	IF(inResult.Result<>eOverallResult.Failed ) THEN
		THIS^.StationBase.RecurringFails.AnyRecurringFails.Counter:=0;
		THIS^.StationBase.RecurringFails.AnyRecurringFails.Reached :=FALSE;
		This^.CompleteStep();
	ELSE
		//collect any recurring fails
		IF NOT THIS^.StationBase.RecurringFails.AnyRecurringFails.Reached THEN 
			THIS^.StationBase.RecurringFails.AnyRecurringFails.Counter := THIS^.StationBase.RecurringFails.AnyRecurringFails.Counter +1;
		END_IF
		THIS^.StationBase.RecurringFails.AnyRecurringFails.Reached:=THIS^.StationBase.RecurringFails.AnyRecurringFails.Counter>=THIS^.StationBase._settings.AnyRecurringFailure;
		

		
	

		
		THIS^.Messenger.OnCondition(THIS^.StationBase.RecurringFails.AnyRecurringFails.Reached)
									   .Build()
									   .Append('(Consecutive failure) The number of any recurring failure count has been reached!')
									   .Append(' Failure code: ')
									   .Append(inResult.ErrorCodes)
  									   .Append(' ')
									   .Append(inResult.Failures)						
									   .As()				   
									   .AsError();
									   
		THIS^.StepCompleteWhen(NOT THIS^.StationBase.RecurringFails.AnyRecurringFails.Reached);			
						   
									   
		IF THIS^.StationBase.RecurringFails.AnyRecurringFails.Reached THEN
			
				
			IF(_dialog.Show()
			   .WithCaption('<#(Consecutive failure) The number of any recurring failure count has been reached!#>')
			   .WithText('<#Please acknowledge recurring failure!#>')
			   .WithOk().Answer = TcoCore.eDialogAnswer.OK) THEN
			   
					THIS^.StationBase.RecurringFails.AnyRecurringFails.Counter:=0;
					THIS^.StationBase.RecurringFails.AnyRecurringFails.Reached :=FALSE;
					THIS^.CompleteStep();
			END_IF; 
		END_IF;
	END_IF;
	

	
	
	
 		    				
    //-------------------------------------
END_IF
END_METHOD

METHOD MonitorSameRecurringFailure
VAR_INPUT
	(*~
	<docu>
		<summary>
			The unique step id definition.
		</summary>			
	</docu>	
	~*)
	inStepID : INT;
		(*~
	<docu>
		<summary>
			The step enable condition.
		</summary>			
	</docu>	
	~*)
	inEnableStep :BOOL;
	inResult : TcoComprehensiveResult;
END_VAR
IF (Step(inStepID,inEnableStep, 'MONITOR SAME RECURRING FAILURE IN SEQUENCE')) THEN
    //-------------------------------------		
	
	IF(inResult.Result<>eOverallResult.Failed ) THEN
		THIS^.StationBase.RecurringFails.SameRecurringFails.Counter:=0;
		THIS^.StationBase.RecurringFails.SameRecurringFails.Reached :=FALSE;
		THIS^.CompleteStep();
	ELSE
	
		//collect same recurring
		IF NOT THIS^.StationBase.RecurringFails.SameRecurringFails.Reached THEN 
			IF THIS^.StationBase.RecurringFails.SameRecurringFails.Result.ErrorCodes = inResult.ErrorCodes AND inResult.ErrorCodes <>';' THEN //if error code not defined ignore
				THIS^.StationBase.RecurringFails.SameRecurringFails.Counter := THIS^.StationBase.RecurringFails.SameRecurringFails.Counter +1;
			END_IF;
			THIS^.StationBase.RecurringFails.SameRecurringFails.Result.ErrorCodes := inResult.ErrorCodes ;
		END_IF;
		
		THIS^.StationBase.RecurringFails.SameRecurringFails.Reached:=THIS^.StationBase.RecurringFails.SameRecurringFails.Counter>=THIS^.StationBase._settings.SameRecurringFailure;

			
		THIS^.Messenger.OnCondition(THIS^.StationBase.RecurringFails.SameRecurringFails.Reached)
									   .Build()
									   .Append('(Consecutive failure) The number of same recurring failure count has been reached!')
									   .Append(' Failure code: ')
									   .Append(inResult.ErrorCodes)
  									   .Append(' ')
									   .Append(inResult.Failures)									   									   
									   .As()				   
									   .AsError();
		
		THIS^.StepCompleteWhen(NOT THIS^.StationBase.RecurringFails.SameRecurringFails.Reached);
	

									   
		IF THIS^.StationBase.RecurringFails.SameRecurringFails.Reached THEN
			IF(_dialog.Show()
			   .WithCaption('<#(Consecutive failure) The number of same recurring failure count has been reached!#>')
			   .WithText('<#Please acknowledge recurring failure!#>')
			   .WithOk().Answer = TcoCore.eDialogAnswer.Ok) THEN
			   
					THIS^.StationBase.RecurringFails.SameRecurringFails.Counter:=0;
					THIS^.StationBase.RecurringFails.SameRecurringFails.Reached :=FALSE;
					THIS^.CompleteStep();
			END_IF; 
		END_IF
	END_IF;
	

	
	
	
 		    				
    //-------------------------------------
END_IF
END_METHOD

PROPERTY StationBase : REFERENCE TO CuBase
GET
VAR
    _station : POINTER TO CUBase;
END_VAR
IF __QUERYPOINTER(Parent, _station) THEN // Check if _Parent is Station001
    StationBase REF= _station^;              // If the check is successful dereference a pointer. simlar to THIS^ or SUPER^
END_IF
END_GET
END_PROPERTY

END_FUNCTION_BLOCK

// ---- Abstractions/TcoCore/TcoTaskedSequencer.TcPOU
FUNCTION_BLOCK PUBLIC ABSTRACT TcoTaskedSequencer EXTENDS TcoCore.TcoSequencerBase
VAR
	{attribute addProperty Name "|[[1]AttributeName]|"}
	{attribute addProperty ToolTip "|[[1]AttributeToolTip]|"}
    _task : TcoInnerTask(THIS^);
    _o    : TcoCore.TcoSequencerObserver(THIS^);	
	{attribute addProperty Name "|[[1]Cycle Time Analitics]|"} 
	_cycleTimeAnalitics:CycleTimeAnalitics;	
	_startCleanCycleTime: TIME;
	_stopCleanCycleTime: TIME;
	_timer_1: TON;
	_timer_2: TON;
END_VAR

Run();

PROPERTY PUBLIC AverageCleanCycleTime : TIME
GET
AverageCleanCycleTime:=_cycleTimeAnalitics.AverageCleanCycle;
END_GET
END_PROPERTY

PROPERTY PUBLIC AverageCycleTime : TIME
GET
AverageCycleTime:=_cycleTimeAnalitics.Average;
END_GET
END_PROPERTY

(*~
	<docu>
		<summary>
			Completes the actually running step, when the `inCondition` parameter is `TRUE`.
			Method is typically called inside a step as the transition method.
		</summary>			
	</docu>	
~*)
METHOD PROTECTED FINAL Await
VAR_INPUT
    (*~
	<docu>
		<summary>
			The condition under which the step is completed.
		</summary>			
	</docu>	
~*)
    inCondition : BOOL;
END_VAR
i_StepCompleteWhen(inCondition := inCondition);
END_METHOD

(*~
	<docu>
		<summary>
			<para>
				Completes the sequencer, and return the sequencer pointer to the first step in the seuqence.
				Method is typically called inside the last step of the sequence.
			</para>
		</summary>			
	</docu>	
~*)
METHOD PROTECTED FINAL CompleteSequence
i_CompleteSequence();

IF _cycleTimeAnalitics.FilterConstant = 0 THEN;
	_cycleTimeAnalitics.FilterConstant:=10;
END_IF;


IF _cycleTimeAnalitics.Average = T#0S THEN
	_cycleTimeAnalitics.Average:=_SequenceElapsedTime;
END_IF
_cycleTimeAnalitics.Average:= (((_cycleTimeAnalitics.FilterConstant-1)*_cycleTimeAnalitics.Average)+_LastCycleTime)/_cycleTimeAnalitics.FilterConstant;

_startCleanCycleTime:=T#0S;
_stopCleanCycleTime:=T#0S;
END_METHOD

(*~
	<docu>
		<summary>
			Completes the execution of the current step and moves the sequencer pointer to the next step in order of execution.
			The call returns `ITcoObjectRestorer` that allows to restore object upon step completition.
		</summary>		
		<returns></returns>	
	</docu>	
~*)
METHOD PROTECTED FINAL CompleteStep : ITcoObjectRestorer
CompleteStep := i_CompleteStep();
END_METHOD

PROPERTY PUBLIC CycleTimeFilterConstant : UINT
GET
CycleTimeFilterConstant:=_cycleTimeAnalitics.FilterConstant;
END_GET
SET // PUBLIC
_cycleTimeAnalitics.FilterConstant:=CycleTimeFilterConstant;
END_SET
END_PROPERTY

(*~
	<docu>
		<summary>
			Main method of the sequener. Custom code needs to be placed here. The sequencer is executed by call of **Instance.Run()** method.
			This method is abstract, and it must be overridden in derived block.
		</summary>
	</docu>
~*)
METHOD PROTECTED  Main : BOOL
END_METHOD

METHOD PUBLIC OnAbort : BOOL
SUPER^.Restore();
END_METHOD

METHOD PUBLIC OnDone : BOOL
END_METHOD

METHOD PUBLIC OnError : BOOL
END_METHOD

METHOD PUBLIC OnStart
_startCleanCycleTime:=T#0S;
_stopCleanCycleTime:=T#0S;
END_METHOD

METHOD pr_Close
VAR_INPUT
END_VAR
_lastClosingCycle := Context.StartCycleCount;

IF _sequencerHasError THEN
    OnSequencerError(_sequencerErrorId);
END_IF

_previousNumberOfStepsInSequence := _numberOfStepsInSequence;
Context.Environment.Messaging.Suspend();

IF _modeController._stepIn.Done THEN
    _modeController._stepIn.Restore();
END_IF

Context.Environment.Messaging.Resume();

_restoringSequence := FALSE;
END_METHOD

METHOD pr_Open
VAR
    _message : STRING(255);
END_VAR
_theOrderOfTheCurrentlyEvaluatedStep := 0;

IF _requestStepActive AND
    _requestedStepId <> (MinStepID - 1) AND
    (_modeController.Mode <> eSequencerMode.StepMode OR _modeController._stepIn.Busy OR _checkStepIdRequestedInStepMode) THEN
    _requestStepCycle := _requestStepCycle + 1;
ELSE
    _requestStepCycle := 0;
END_IF

IF _requestStepCycle > 1 AND NOT _sequencerHasError THEN
    _sequencerErrorId        := eSequencerError.StepWithRequestedIdDoesNotExists;
    _message                 := CONCAT('REQUESTED STEP_ID: ', INT_TO_STRING(_requestedStepId));
    _message                 := CONCAT(_message, ' DOES NOT EXIST');
    _currentStep.Description := _message;
    _currentStep.Status      := eStepStatus.Error;
    THIS^.Messenger.Post(_message, eMessageCategory.ProgrammingError);
    _sequencerHasError := TRUE;
END_IF

IF _StepIdUniquenessControlState = eStepIdUniquenessControlState.NotYetStarted OR
    _StepIdUniquenessControlState = eStepIdUniquenessControlState.Requested THEN
    _StepIdUniquenessControlState := eStepIdUniquenessControlState.Started;
END_IF;

_restoringSequence := FALSE;

_lastOpeningCycle := Context.StartCycleCount;
;
END_METHOD

(*~
	<docu>
		<summary>
			Terminates the currently executed step and set the sequencer's pointer to the step with Id that corresponds to ```inRequestedStepID``` parameter.
			When the order of the requested step is higher than the order of the currently finished step (the requested step is "after" the current one)
			the requested step is started in the same context cycle.
			When the order of the requested step is lower than the order of the currently finished step (the requested step is "before" the current one)
			the requested step is started in the next context cycle.
			If the requested step is not found even in the next context cycle, the sequencer enters error state ```StepWithRequestedIdDoesNotExists```.
			<para>
				See <see cref="TcoCore.eSequencerError"/> for detailed description.
			</para>
		</summary>
	</docu>
~*)
METHOD PROTECTED FINAL RequestStep : ITcoSequencer
VAR_INPUT
    (*~
		<docu>
			<summary>
				StepId of the step to be executed.
			</summary>
		</docu>
	~*)
    inRequestedStepID : INT := MinStepID - 1;
END_VAR
VAR
    _message : STRING(254);
END_VAR
RequestStep := i_RequestStep(inRequestedStepID := inRequestedStepID);
END_METHOD

(*~
	<docu>
		<summary>
			This method resets the sequencer cycle time . 
				Method is typically called before starting the sequence(e.g.in ground position task) .
		</summary>		
		<returns></returns>	
	</docu>	
~*)
METHOD PUBLIC ResetCycleTime
VAR_INPUT
END_VAR

_cycleTimeAnalitics.Average:=T#0S;
_cycleTimeAnalitics.AverageCleanCycle:=T#0S;
END_METHOD

METHOD PRIVATE ResetTimers
VAR_INPUT
END_VAR
_timer_1.IN:=FALSE;
_timer_2.IN:=FALSE;
END_METHOD

(*~
	<docu>
		<summary>
			<para>
				This method resets the sequencer. 
				Method is typically called before starting the sequence or after error has occured in the sequence.
			</para>
		</summary>			
	</docu>	
~*)
METHOD PUBLIC Restore : ITcoRestorable
SUPER^.Restore();
Task.Restore();
END_METHOD

(*~
	<docu>
		<summary>
			<para>
				Ensures calling the Open(), Main() and Close() methods in the desired order.
				This method is final, so it cannot be overloaded. The **Instance.Run()** needs to be called cyclically inside the appropriate context.
			</para>
		</summary>			
	</docu>	
~*)
METHOD PUBLIC FINAL Run
VAR
    _message : STRING;
END_VAR
IF (_task.Execute()) THEN
    THIS^.pr_Open();
    THIS^.Observer := _o;
    THIS^.Main();
    THIS^.pr_Close();
END_IF;
END_METHOD

(*~
	<docu>
		<summary>
			This method s used to start the clean cycle time measurement . 
				Method is typically called at the beggining of the sequence(e.g.in automat sequence) .
		</summary>		
		<returns></returns>	
	</docu>	
~*)

METHOD PUBLIC StartCleanCycleTime
VAR_INPUT
END_VAR
_stopCleanCycleTime:=t#0s;
_startCleanCycleTime:=_SequenceElapsedTime;
END_METHOD

METHOD PROTECTED Step : BOOL
VAR_INPUT
    (*~
	<docu>
		<summary>
			StepId of the current step.
			<remarks>			
				<note type="important">
					This number must be unique throughout the complete sequence.
					It must be a constant or numerical literal and it must not change during the life-time of the sequencer. 
				</note>
			</remarks>
		</summary>		
	</docu>	
~*)
    inStepID : INT;
    (*~
	<docu>
		<summary>
			If this value is false, step body is not executed and execution is moved to the next enabled step.
		</summary>				
	</docu>	
~*)
    inEnabled : BOOL;
    (*~
	<docu>
		<summary>
			Step description text.
		</summary>				
	</docu>	
~*)
    inStepDescription : STRING(254);
END_VAR
Step := i_Step(inStepID := inStepID, inEnabled := inEnabled, inStepDescription := inStepDescription);
END_METHOD

(*~
	<docu>
		<summary>
			Completes the actually running step, when the `inCondition` parameter is `TRUE`.
			Method is typically called inside a step as the transition method.
		</summary>			
	</docu>	
~*)
METHOD PROTECTED FINAL StepCompleteWhen
VAR_INPUT
    (*~
	<docu>
		<summary>
			The condition under which the step is completed.
		</summary>			
	</docu>	
~*)
    inCondition : BOOL;
END_VAR
i_StepCompleteWhen(inCondition := inCondition);
END_METHOD

(*~
	<docu>
		<summary>
			This method s used to stop the clean cycle time measurement . 
				Method is typically called at the end of the sequence(e.g.in automat sequence )  .
		</summary>		
		<returns></returns>	
	</docu>	
~*)

METHOD PUBLIC StopCleanCycleTime
VAR_INPUT
END_VAR

VAR
	cleanCycleTime: TIME;
END_VAR
_stopCleanCycleTime:=_SequenceElapsedTime;

cleanCycleTime:=T#0S;
IF _stopCleanCycleTime>_startCleanCycleTime THEN
	cleanCycleTime:=_stopCleanCycleTime-_startCleanCycleTime;
 END_IF;

IF _cycleTimeAnalitics.FilterConstant = 0 THEN;
	_cycleTimeAnalitics.FilterConstant:=10;
END_IF;


IF _cycleTimeAnalitics.AverageCleanCycle = T#0S THEN
	_cycleTimeAnalitics.AverageCleanCycle:=_stopCleanCycleTime;
END_IF
_cycleTimeAnalitics.AverageCleanCycle:= (((_cycleTimeAnalitics.FilterConstant-1)*_cycleTimeAnalitics.AverageCleanCycle)+cleanCycleTime)/_cycleTimeAnalitics.FilterConstant;
END_METHOD

PROPERTY Task : REFERENCE TO TcoTask
GET
Task REF= _task;
END_GET
END_PROPERTY

METHOD PUBLIC FINAL Timer_1 : BOOL
VAR_INPUT
	Condition : BOOL;
	PT : TIME;
END_VAR
_timer_1(IN:= Condition  and  not IsFreshState, PT:=PT);
Timer_1 := _timer_1.Q;
END_METHOD

METHOD PUBLIC FINAL Timer_2 : BOOL
VAR_INPUT
	Condition : BOOL;
	PT : TIME;
END_VAR
_timer_2(IN:= Condition and not IsFreshState, PT:=PT);
Timer_2 := _timer_2.Q;
END_METHOD

END_FUNCTION_BLOCK

// ---- Abstractions/TcoCore/TcoInnerTask.TcPOU
FUNCTION_BLOCK TcoInnerTask EXTENDS TcoCore.TcoTask

(*~
	<docu>
		<summary>
			Executes when task is aborted.
		</summary>			
	</docu>	
~*)
METHOD PROTECTED OnAbort
ParentSequencer.OnAbort();
END_METHOD

(*~
	<docu>
		<summary>
			Executes when task reaches the ```Done``` state .
		</summary>			
	</docu>	
~*)
METHOD PROTECTED OnDone
ParentSequencer.OnDone();
END_METHOD

(*~
	<docu>
		<summary>
			Executes when task reaches the ```Error``` state.
			<para>
				Do not confuse with <see cref="PlcDocu.TcoCore.TcoTask.WhileError()"/>, that is called cyclically until '''Error''' state is left.
			</para>
		</summary>			
	</docu>	
~*)
METHOD PROTECTED OnError
ParentSequencer.OnError();
END_METHOD

METHOD PROTECTED OnStart
ParentSequencer.OnStart();
END_METHOD

PROPERTY PRIVATE ParentSequencer : REFERENCE TO TcoTaskedSequencer
GET
VAR
	_sequencer : POINTER TO TcoTaskedSequencer;
END_VAR
IF __QUERYPOINTER(Parent, _sequencer) THEN // Check if _Parent is Station001
    ParentSequencer REF= _sequencer^;              // If the check is successful dereference a pointer. simlar to THIS^ or SUPER^
END_IF
END_GET
END_PROPERTY

END_FUNCTION_BLOCK

// ---- Abstractions/CUBase/Tasks/CUBaseGround.TcPOU
FUNCTION_BLOCK ABSTRACT CUBaseGround EXTENDS TcoTaskedSequencer
VAR
	_groundDone : BOOL;
END_VAR

METHOD INTERNAL CancelGround
_groundDone := FALSE;
END_METHOD

PROPERTY GroundDone : BOOL
GET
GroundDone := _groundDone;
END_GET
END_PROPERTY

END_FUNCTION_BLOCK

// ---- Abstractions/TcoCore/TcoTaskedService.TcPOU
FUNCTION_BLOCK PUBLIC ABSTRACT TcoTaskedService EXTENDS TcoCore.TcoTask
VAR
	
END_VAR

(*~
	<docu>
		<summary>
			Main method of the sequener. Custom code needs to be placed here. The sequencer is executed by call of **Instance.Run()** method.
			This method is abstract, and it must be overridden in derived block.
		</summary>
	</docu>
~*)
METHOD PROTECTED ABSTRACT Main : BOOL
END_METHOD

(*~
	<docu>
		<summary>
			<para>
				Ensures calling the Open(), Main() and Close() methods in the desired order.
				This method is final, so it cannot be overloaded. The **Instance.Run()** needs to be called cyclically inside the appropriate context.
			</para>
		</summary>			
	</docu>	
~*)
METHOD PUBLIC FINAL Run
VAR
    _message : STRING;
END_VAR
IF (THIS^.Execute()) THEN
    THIS^.Main();    
END_IF;
END_METHOD

PROPERTY Task : REFERENCE TO TcoTask
GET
Task REF= THIS^;
END_GET
END_PROPERTY

END_FUNCTION_BLOCK

// ---- Abstractions/CUBase/Tasks/CUBaseRecover.TcPOU
FUNCTION_BLOCK ABSTRACT CUBaseRecover EXTENDS TcoTaskedSequencer
VAR
	_done:BOOL;

END_VAR

PROPERTY Done : bool
GET
Done := _done;
END_GET
END_PROPERTY

METHOD PUBLIC OnStart
_done:=FALSE;
END_METHOD

PROPERTY StationBase : REFERENCE TO CuBase
GET
VAR
    _station : POINTER TO CuBase;
END_VAR
IF __QUERYPOINTER(Parent, _station) THEN // Check if _Parent is Station001
    StationBase REF= _station^;              // If the check is successful dereference a pointer. simlar to THIS^ or SUPER^
END_IF
END_GET
END_PROPERTY

END_FUNCTION_BLOCK

// ---- Abstractions/CUBase/Tasks/CUBaseSuspend.TcPOU
FUNCTION_BLOCK ABSTRACT CUBaseSuspend EXTENDS TcoTaskedSequencer
VAR
	_done:BOOL;

END_VAR

PROPERTY Done : bool
GET
Done := _done;
END_GET
END_PROPERTY

METHOD PUBLIC OnStart
_done:=FALSE;
END_METHOD

PROPERTY StationBase : REFERENCE TO CuBase
GET
VAR
    _station : POINTER TO CuBase;
END_VAR
IF __QUERYPOINTER(Parent, _station) THEN // Check if _Parent is Station001
    StationBase REF= _station^;              // If the check is successful dereference a pointer. simlar to THIS^ or SUPER^
END_IF
END_GET
END_PROPERTY

END_FUNCTION_BLOCK

// ---- Technology/CU00x/Manual/CU00xManualTask.TcPOU
FUNCTION_BLOCK CU00xManualTask EXTENDS TcoTaskedService IMPLEMENTS ICUTask
VAR
END_VAR

Run();

(*~
	<docu>
		<summary>
			Main method of the sequener. Custom code needs to be placed here. The sequencer is executed by call of **Instance.Run()** method.
			This method is abstract, and it must be overridden in derived block.
		</summary>
	</docu>
~*)
METHOD PROTECTED Main : BOOL
Messenger.Notify('Running manual mode');
// Station.Components.OUT1.Service();
// Station.Components.OUT2.Service();
// Station.Components.OUT3.Service();
END_METHOD

METHOD PROTECTED OnStart
Station.AutomatTask.Restore();
Station.GroundTask.Restore();
Station.GroundTask.CancelGround();
END_METHOD

PROPERTY Station : REFERENCE TO CU00x
GET
VAR
    _station : POINTER TO CU00x;
END_VAR
IF __QUERYPOINTER(Parent, _station) THEN // Check if _Parent is Station001
    Station REF= _station^;              // If the check is successful dereference a pointer. simlar to THIS^ or SUPER^
END_IF
END_GET
END_PROPERTY

END_FUNCTION_BLOCK

// ---- Technology/CU00x/Ground/CU00xGroundTask.TcPOU
FUNCTION_BLOCK CU00xGroundTask EXTENDS CUBaseGround IMPLEMENTS ICUTask

Run();

METHOD DataEntityDiscard
VAR_INPUT	
	inStepID : INT;
	EntityId : STRING(255);
END_VAR
IF (Step(inStepID, TRUE, 'DISCARD ENTITY')) THEN	
    //-------------------------------------		
	IF(Station.ProcessDataManager.Exists(EntityId).Done) THEN
		IF(Station.ProcessDataManager._idExistsTask.Exists) THEN
			StepCompleteWhen(THIS^.Station.EntityFlowDiscard(EntityId, Station.ProcessDataManager.Data.CU00x.Header).Done);
		ELSE
			CompleteStep();
		END_IF
	END_IF;					   		    				
    //-------------------------------------
END_IF
END_METHOD

(*~
	<docu>
		<summary>
			Main method of the sequener. Custom code needs to be placed here. The sequencer is executed by call of **Instance.Run()** method.
			This method is abstract, and it must be overridden in derived block.
		</summary>
	</docu>
~*)
METHOD PROTECTED Main : BOOL
IF (Step(100, TRUE, 'STOPPING OTHER MODES')) THEN
	Station.AutomatTask.ResetCycleTime();//here we can reset averages values of CT
	Station.AutomatTask.Restore();
	Station.ManualTask.Restore();
	Station.ProcessDataManager.Restore();
	Station.AutomatTask.HideAllDialogs();
	Station.GroupInspection.Restore();// hide all dialogs 
    StepCompleteWhen(TRUE);
END_IF

IF (Step(200, TRUE, 'STOPPING OTHER MODES')) THEN	
//	---------------------------------------------------
	
	Station.AutomatTask.ResetCycleTime();
	Station.ProductionPlanerTask.Restore();
	
	Messenger.Info('INFO MESSAGE');
	
    StepCompleteWhen(THIS^._currentStep.Duration > T#500MS);
//	---------------------------------------------------
END_IF

DataEntityDiscard(5000, THIS^.Station.ProcessDataManager.Data._EntityId);

IF (Step(10000, TRUE, 'LAST STEP')) THEN	
	//---------------------------------------------------
	_groundDone := TRUE;
	THIS^._task.DoneWhen(_groundDone);
	//---------------------------------------------------
END_IF
END_METHOD

METHOD PUBLIC OnStart
SUPER^.OnStart();
Station.AutomatTask.Restore();
Station.ManualTask.Restore();
Station.GroundTask.CancelGround();
END_METHOD

PROPERTY Station : REFERENCE TO CU00x
GET
VAR
    _station : POINTER TO CU00x;
END_VAR
IF __QUERYPOINTER(Parent, _station) THEN // Check if _Parent is Station001
    Station REF= _station^;              // If the check is successful dereference a pointer. simlar to THIS^ or SUPER^
END_IF
END_GET
END_PROPERTY

END_FUNCTION_BLOCK

// ---- Technology/CU00x/Automat/CU00xAutomatTask.TcPOU
FUNCTION_BLOCK CU00xAutomatTask EXTENDS CUBaseAutomat IMPLEMENTS ICUTask
VAR

    _missingProcessSettingMessage : TcoCore.TcoMessenger(THIS^);
    _paralellTask : CU00xAutomatParalell_1_Task(THIS^, TcoCore.eRestoreMode.None);

    _sb : TcoCore.StringBuilder;

    _customizedContentInput : CU00xDialogContent(THIS^);
END_VAR

VAR
    _dataLoadProcessSettings : BOOL;
    _dataLoadProcessSettingsByPlaner : BOOL;
    _dataCreateNew : BOOL;
    _dataOpen : BOOL;
    _dataClose : BOOL;
    _dataFinalize : BOOL;
    _continueRestore : BOOL;
    _loop : BOOL;
    _inspectionResult : BOOL;
    _inspectionDimensionResult : REAL;
    _reqKey : STRING;
    _reqAssignedValue : STRING;
    _inspectorSingleExamples : BOOL;
    _inspectorGroupExamples : BOOL;
	_dialogExamples : BOOL;

END_VAR

Run();

(*~
	<docu>
		<summary>
			Loads technology settings from the current technology set into this controlled unit.
			The `StationProcessDataManager.Data` is populated by data from process settings.						
		</summary>
	</docu>
~*)
METHOD DataLoadProcessSettings : BOOL
VAR_INPUT
	inStepID : INT;
END_VAR

VAR
	_ans: TcoCore.eDialogAnswer;
END_VAR
IF (Step(inStepID, _dataLoadProcessSettings, 'LOAD PROCESS SETTING')) THEN
    //-------------------------------------
	
	THIS^._missingProcessSettingMessage.OnCondition(Station.Technology.ProcessSettings.Data._EntityId = '')
									   .Build()
									   .Append('No process data. Please load setting')
									   .As()				   
									   .AsError()
									   .Pin();
					   
				   
	IF(Station.Technology.ProcessSettings.Data._EntityId <> '' (*AND NOT THIS^._missingProcessSettingMessage.Pinned*)) THEN
		IF(Station.Technology.ProcessSettings.Read(Station.Technology.ProcessSettings.Data._EntityId).Done) THEN
			Station.ProcessDataManager.Data := Station.Technology.ProcessSettings.Data;
			Station.ProcessDataManager.Data.EntityHeader.RecipeCreated := Station.Technology.ProcessSettings.Data._Created;
			Station.ProcessDataManager.Data.EntityHeader.RecipeLastModified  := Station.Technology.ProcessSettings.Data._Modified;
			Station.ProcessDataManager.Data.EntityHeader.Recipe  := Station.Technology.ProcessSettings.Data._EntityId;				
			CompleteStep();

		END_IF;	
	ELSE
		_ans:=_dialog.Show()
			.WithImage('d:\MTS\Develop\TcOpenGroup\TcOpen\assets\logo\TcOpenWide.png',400,600)	
	       .WithCaption('<#Process data not selected#>')
		   .WithText('<#Would you like to load default settings?#>')
		   .WithYesNoCancel().Answer;
		IF(_ans=TcoCore.eDialogAnswer.Cancel) THEN
			this^.Restore();
		END_IF
		IF( _ans= TcoCore.eDialogAnswer.Yes) THEN
		   
		   	Station.Technology.ProcessSettings.Data._EntityId := 'default';
		END_IF; 

			
	END_IF		    				
    //-------------------------------------
END_IF
END_METHOD

(*~
	<docu>
		<summary>
			Loads process settings from the current process set into this controlled unit.
			The `StationProcessDataManager.Data` is populated by data from process settings.						
		</summary>
	</docu>
~*)
METHOD DataLoadProcessSettingsByPlaner : BOOL
VAR_INPUT
	inStepID : INT;
END_VAR
IF (Step(inStepID, _dataLoadProcessSettingsByPlaner, 'LOAD PROCESS SETTING BY THE PRODUCTION PLANER')) THEN
    //-------------------------------------


								   
	 IF Station.ProductionPlanerTask.Invoke().Done	AND_THEN(Station.ProductionPlanerTask.RequiredProcessSettingsId <> '') THEN
		
		IF NOT Station.ProductionPlanerTask.ProductionPlanCompleted and_then (Station.Technology.ProcessSettings.Read(Station.ProductionPlanerTask.RequiredProcessSettingsId).Done)
			 THEN
			Station.ProcessDataManager.Data := Station.Technology.ProcessSettings.Data;
			Station.ProcessDataManager.Data.EntityHeader.RecipeCreated := Station.Technology.ProcessSettings.Data._Created;
			Station.ProcessDataManager.Data.EntityHeader.RecipeLastModified  := Station.Technology.ProcessSettings.Data._Modified;
			Station.ProcessDataManager.Data.EntityHeader.Recipe  := Station.Technology.ProcessSettings.Data._EntityId;				
			CompleteStep();
			Station.ProductionPlanerTask.Restore();
		END_IF;
	ELSIF  Station.ProductionPlanerTask.ProductionPlanIsEmpty THEN
		IF (_dialog.Show()
	       .WithCaption('<#Production planer#>')
		   .WithText('<#Production planer is empty!#>')
			.WithOk().Answer = TcoCore.eDialogAnswer.OK) THEN;
			;// Production plan comleted , here you can write diferent scenario ( leave it with current state , provide ground etc)	 
	
		 	//Station.GroundTask.Task.Invoke();
		   
		End_if;
	
	ELSIF  Station.ProductionPlanerTask.ProductionPlanCompleted THEN
		IF (_dialog.Show()
	       .WithCaption('<#Production planer#>')
		   .WithText('<#Production planer completed required plan!#>')
			.WithOk().Answer = TcoCore.eDialogAnswer.OK) THEN;
			;// Production plan comleted , here you can write diferent scenario ( leave it with current state , provide ground etc)	 
	
		 	//Station.GroundTask.Task.Invoke();
		   
		End_if;

			
	END_IF		    				
    //-------------------------------------
END_IF
END_METHOD

METHOD DialogExamples
VAR_INPUT
		inStepID : INT;
END_VAR
IF (Step(inStepID, TRUE, 'DIALOG EXAMPLE ')) THEN
//-------------------------------------
		_dialog.Show()
            .WithType(eDialogType.Question)
            .WithYesNo()
            .WithCaption('Hey')
            .WithText('Do we go ahead ');

        IF (_dialog.Answer = TcoCore.eDialogAnswer.Yes) THEN
            CompleteStep();
        END_IF;

        IF (_dialog.Answer = TcoCore.eDialogAnswer.No) THEN
            ;
        END_IF;

//-------------------------------------
END_IF;

IF (Step(inStepID+10, TRUE, 'DIALOG EXAMPLE WIT IMAGE')) THEN
//-------------------------------------
		_dialog.Show()
            .WithType(eDialogType.Question)
            .WithYesNo()
			.WithImage('D:\MTS\Develop\TcOpenGroup\TcOpen\assets\logo\TcOpenLogo.png',400,600)
            .WithCaption('Hey 1')
            .WithText('Do we go ahead ?');

        IF (_dialog.Answer = TcoCore.eDialogAnswer.Yes) THEN
            CompleteStep();
        END_IF;

        IF (_dialog.Answer = TcoCore.eDialogAnswer.No) THEN
            ;
        END_IF;

//-------------------------------------
END_IF;


IF (Step(inStepID+20, TRUE, 'DIALOG EXAMPLE WITH CLOSE FROM PLC')) THEN
//-------------------------------------
		_dialog.ShowWithExternalClose(inOkAnswerSignal:=FALSE , inYesAnswerSignal:= CurrentStep.Duration>T#2000MS, inNoAnswerSignal:= FALSE, inCancelAnswerSignal:= FALSE)
		    .WithType(eDialogType.Info)
            .WithYesNoCancel()
            .WithCaption('Hey')
            .WithText('Do you wana retry it? Yes answer will be set in 4 sec?');

        IF (_dialog.Answer = TcoCore.eDialogAnswer.Yes) THEN
            CompleteStep();
        END_IF;

      

//-------------------------------------
END_IF;

IF (Step(inStepID+30, TRUE, 'CUSTOMIZED DIALOG EXAMPLE WITH CLOSE FROM PLC ')) THEN
//-------------------------------------
			 _dialogCustomized.ShowWithExternalClose(inOption1AnswerSignal:=FALSE,inOption2AnswerSignal:=FALSE, inOption3AnswerSignal:=CurrentStep.Duration>T#4000MS,inOption4AnswerSignal:=FALSE)
            
            .WithOption1('This is Option1=>retry')
			  .WithOption2('This is Option2=>first step')
			    .WithOption3('This is Option3 =>continue and finish in 4s')
			.WithImage('D:\MTS\Develop\TcOpenGroup\TcOpen\assets\logo\TcOpenWide.png',500,500)
            .WithCaption('Hey')
            .WithText('What we are going to do.');
            
		
           
	
			IF (_dialogCustomized.Answer = TcoCore.eCustomizedDialogAnswer.Option3) THEN
				CompleteStep();
			END_IF;

//-------------------------------------
END_IF;

IF (Step(inStepID+40, TRUE, 'INPUT DIALOG EXAMPLE  REQURED FIELDS TO INPUT DATA')) THEN
//-------------------------------------
		_dialogWithInput.Show(refContent:=_customizedContentInput)
            .WithType(eDialogType.Question)
            .WithYesNo()
            .WithCaption('Hey wana set data')
            .WithText('Do you realy want to sent data to ....?');
                
		IF (_dialogWithInput.Answer = TcoCore.eInputDialogAnswer.Yes) THEN
				CompleteStep();
			//by yes or (ok) option data are confirmed and transfered to plc (_customizedContentInput)
		ELSIF (_dialogWithInput.Answer = TcoCore.eInputDialogAnswer.No) THEN
			// data in struct '_customizedContentInput' remains same as before
 		END_IF;
		

//-------------------------------------
END_IF;
IF (Step(inStepID+50, TRUE, 'INPUT DIALOG EXAMPLE WITH WEB CONTENT AND REQURED FIELDS TO INPUT DATA')) THEN
//-------------------------------------
		_dialogWithInput.Show(refContent:=_customizedContentInput)
            .WithType(eDialogType.Question)
            .WithOk()
			.WithImage('https://github.com/TcOpenGroup',400,600)
            .WithCaption('Hey wana set data')
            .WithText('Do you realy want to sent data to ....?');
			
                
		IF (_dialogWithInput.Answer = TcoCore.eInputDialogAnswer.OK) THEN
			CompleteStep();
			
		END_IF;

//-------------------------------------
END_IF;
END_METHOD

METHOD GroupedExample
VAR_INPUT
		inStepID : INT;
END_VAR
IF (Step(inStepID, TRUE, 'MULTI ANALOGUE INSPECTIONS PART 1 WITH WEB CONTENT')) THEN
//-------------------------------------
		Station.GroupInspection
		.WithCoordinator(THIS^)
		.Act();
		Station.GroupInspection.Inspect(Station.ProcessDataManager.Data.CU00x.Dim_Inspector_1.WithCoordinator(THIS^).Inspect(0));	
		Station.GroupInspection.Inspect(Station.ProcessDataManager.Data.CU00x.Dim_Inspector_2.WithCoordinator(THIS^).Inspect(0));	
		Station.GroupInspection.Inspect(Station.ProcessDataManager.Data.CU00x.Dim_Inspector_3.WithCoordinator(THIS^).Inspect(0));	
		Station.GroupInspection.Inspect(Station.ProcessDataManager.Data.CU00x.Dim_Inspector_4.WithCoordinator(THIS^).Inspect(0));	
		Station.GroupInspection.Inspect(Station.ProcessDataManager.Data.CU00x.Dim_Inspector_5.WithCoordinator(THIS^).Inspect(0));	
		Station.GroupInspection.Inspect(Station.ProcessDataManager.Data.CU00x.Dim_Inspector_6.WithCoordinator(THIS^).Inspect(1));	
		Station.GroupInspection.Inspect(Station.ProcessDataManager.Data.CU00x.Dim_Inspector_7.WithCoordinator(THIS^).Inspect(0));	
		Station.GroupInspection.Inspect(Station.ProcessDataManager.Data.CU00x.Dim_Inspector_8.WithCoordinator(THIS^).Inspect(0));	
		Station.GroupInspection.Inspect(Station.ProcessDataManager.Data.CU00x.Dim_Inspector_9.WithCoordinator(THIS^).Inspect(0));	
		Station.GroupInspection.Inspect(Station.ProcessDataManager.Data.CU00x.Dim_Inspector_10.WithCoordinator(THIS^).Inspect(0));	
	
		
		Station.GroupInspection.UpdateComprehensiveResult(Station.ProcessDataManager.Data.EntityHeader.Results)	
		.Instruct('Something is wrong 1')
		.InstructWithImage('https://github.com/TcOpenGroup/TcOpen/blob/dev/README.md',400,600)	
		.OnFail()
		.Dialog(inStepID+10);			
//-------------------------------------
END_IF;
IF (Step(inStepID+10, TRUE, 'MULTI ANALOGUE INSPECTIONS PART 2 WITH INSTRUCTION AND DESCRIPTION')) THEN
//-------------------------------------
		Station.GroupInspection
		.WithCoordinator(THIS^)
		.Act();
		Station.GroupInspection.Inspect(Station.ProcessDataManager.Data.CU00x.Dim_Inspector_11.WithCoordinator(THIS^).Inspect(0));	
		Station.GroupInspection.Inspect(Station.ProcessDataManager.Data.CU00x.Dim_Inspector_12.WithCoordinator(THIS^).Inspect(0));	
		Station.GroupInspection.Inspect(Station.ProcessDataManager.Data.CU00x.Dim_Inspector_13.WithCoordinator(THIS^).Inspect(0));	
		Station.GroupInspection.Inspect(Station.ProcessDataManager.Data.CU00x.Dim_Inspector_14.WithCoordinator(THIS^).Inspect(0));	
		Station.GroupInspection.Inspect(Station.ProcessDataManager.Data.CU00x.Dim_Inspector_15.WithCoordinator(THIS^).Inspect(0));	
		Station.GroupInspection.Inspect(Station.ProcessDataManager.Data.CU00x.Dim_Inspector_16.WithCoordinator(THIS^).Inspect(1));	
		Station.GroupInspection.Inspect(Station.ProcessDataManager.Data.CU00x.Dim_Inspector_17.WithCoordinator(THIS^).Inspect(0));	
		Station.GroupInspection.Inspect(Station.ProcessDataManager.Data.CU00x.Dim_Inspector_18.WithCoordinator(THIS^).Inspect(0));	
		Station.GroupInspection.Inspect(Station.ProcessDataManager.Data.CU00x.Dim_Inspector_19.WithCoordinator(THIS^).Inspect(0));	
		Station.GroupInspection.Inspect(Station.ProcessDataManager.Data.CU00x.Dim_Inspector_20.WithCoordinator(THIS^).Inspect(0));	
	
		
		Station.GroupInspection.UpdateComprehensiveResult(Station.ProcessDataManager.Data.EntityHeader.Results)	
		.WithDescription()
		.Instruct('Something is wrong 2')
		.OnFail()
		.Dialog(inStepID+20);			
//-------------------------------------
END_IF;

IF (Step(inStepID+20, TRUE, 'DONE')) THEN
//-------------------------------------
		CompleteStep();
//-------------------------------------
END_IF;
END_METHOD

(*~
	<docu>
		<summary>
			Main method of the sequener. Custom code needs to be placed here. The sequencer is executed by call of **Instance.Run()** method.
			This method is abstract, and it must be overridden in derived block.
		</summary>
	</docu>
~*)
METHOD PROTECTED Main : BOOL
(*

	OPENING DATA OPERATIONS
	Following methods provide process data manipulation for this controlled unit.
	Remove `IF` statement and comment or uncomment according to your need.
*)
// Loads process settings. 
// Typically used in the first station of the technology to load process settings that will be used trough out the production
IF (_dataLoadProcessSettings) THEN
    THIS^.DataLoadProcessSettings(100);
END_IF;

// Loads process settings via produciton planer. 
// Typically used in the first station of the technology to load process settings that will be used trough out the production 
// .......
IF (_dataLoadProcessSettingsByPlaner) THEN
    THIS^.DataLoadProcessSettingsByPlaner(110);
END_IF;

(*

		
		This step we would like to star cycle time (e.g. we want to exclude loading data from clean cycle time )		
*)
IF (Step(150, TRUE, '<#START MEASURE CT TRIGGER#>')) THEN
    //-------------------------------------    
    StartCleanCycleTime();
    StepCompleteWhen(TRUE);
    //-------------------------------------
END_IF

// Creates new data entity (new part/item) 
// Typically used in the first station of the technology to create new document/record to be persited in the repository.
// Sets the status of the entity to 'InProgress'
IF (_dataCreateNew) THEN
	IF (Step(160, TRUE, 'CREATE ENTIY ID')) THEN
		//-------------------------------------    
		Station.ProcessDataManager.Data._EntityId := ULINT_TO_STRING(Context.RealTimeClock.TickClock());
	
		StepCompleteWhen(Station.ProcessDataManager.Data._EntityId<>'');
		//-------------------------------------
	END_IF
    THIS^.DataEntityCreateNew(200, Station.ProcessDataManager.Data._EntityId, Header := Station.ProcessDataManager.Data.CU00x.Header);
END_IF;

// Populates the information in the data header of this controlled unit (operation start time stamp, user info, etc)
// Typically used prior to starting operation within a controlled unit.
IF (_dataOpen) THEN
    THIS^.DataEntityOpen(300,
        30000,
        Station.ProcessDataManager.Data._EntityId,
        Station.ProcessDataManager.Data.CU00x.Header);
END_IF;


// Handle user defined carier id
// Typically used in the first station of the technology to assign user defined carier ID  instead of raw unique id(RfidChip....)

(*

		STEPS OF THE SEQUENCE
		Here we would place steps to perfom the operations of this controlled unit.

*)



IF (Step(900, TRUE, 'SINGLE INSPECTION')) THEN
    //-------------------------------------    
	Station.ProcessDataManager.Data.CU00x.BoltPresenceInspector.Data.FailureDescription:='BoltPresenceInspector error';
    Station.ProcessDataManager.Data.CU00x.BoltPresenceInspector.WithCoordinator(THIS^)
        .Inspect(_inspectionResult)
        .UpdateComprehensiveResult(Station.ProcessDataManager.Data.EntityHeader.Results)
        .OnFail().CarryOn();
    //-------------------------------------
END_IF

IF (Step(910, TRUE, 'SINGLE ANALOGUE INSPECTION')) THEN
    //-------------------------------------    
		Station.ProcessDataManager.Data.CU00x.BoltDimensionPresenceInspector.Data.FailureDescription:='BoltDimensionPresenceInspector error';

    Station.ProcessDataManager.Data.CU00x.BoltDimensionPresenceInspector.WithCoordinator(THIS^)
        .Inspect(_inspectionDimensionResult)
        .UpdateComprehensiveResult(Station.ProcessDataManager.Data.EntityHeader.Results)
        .OnFail().CarryOn();
    //-------------------------------------
END_IF


//dialog usage examples
IF _dialogExamples THEN
	DialogExamples(1000);
END_IF;

//single inspexction usage
IF _inspectorSingleExamples THEN
	SingleExample(1100);
END_IF;

// grouped usage of isnpectors
IF _inspectorGroupExamples THEN
	GroupedExample(1200);
END_IF;


IF (Step(2000, true, 'START PARALELL TASK')) THEN
    //-------------------------------------    
    StepCompleteWhen(_paralellTask.Task.Invoke().Busy);
    //-------------------------------------
END_IF

(*

		RECOVERY STEPS
		This step and the following steps should bring the controlled unit in a state from which 
		the sequence can be safely restarted from the beginning of the this sequencer. 		
*)
IF (Step(RESTORE_STEP_ID, TRUE, 'FIRST RESTORE STEP')) THEN
    //-------------------------------------
    StepCompleteWhen(_continueRestore);
    //-------------------------------------	
END_IF

(*

		
		This step we would save cycle time value (e.g. we not include saving data into cycle time )
		
*)
IF (Step(2150, TRUE, 'STOP MEASURE CT TRIGGER')) THEN
    //-------------------------------------    
    StopCleanCycleTime();
    StepCompleteWhen(TRUE);
    //-------------------------------------
END_IF

(*

	CLOSING DATA OPERATIONS
	Following methods provide process data manipulation for this controlled unit.
	Comment or uncomment according to your need.
*)
// Populates the information in the data header of this controlled unit (operations end time stamp, user info, etc)
// Typically used after all steps within the controlled unit are completed.
IF (_dataClose) THEN
    THIS^.DataEntityClose(5000, eDataEntityInvokeType.InvokeAndWaitDone, Station.ProcessDataManager.Data.CU00x.Header);
END_IF;

// Populates the information in the data header of this controlled unit (operations end time stamp, user info, etc)
// Typically used after all operation on the technology are completed.
// Input parameter eDataEntityInvokeType.InvokeOnly is used for speed up cycle(TRUE)
IF (_dataFinalize) THEN
    THIS^.DataEntityFinalize(5500, eDataEntityInvokeType.InvokeOnly, Station.ProcessDataManager.Data.CU00x.Header);
END_IF;

IF (Step(10000, TRUE, 'WAIT FOR PARALELL TASK TO FINISH')) THEN
    //-------------------------------------
    StepCompleteWhen(_paralellTask.Task.Done);

    IF _paralellTask.Task.Done THEN
        _paralellTask.Restore();
    END_IF
    //-------------------------------------	
END_IF

IF (Step(20000, _dataClose, 'WAIT FOR IF DATA FINALIZE IS DONE')) THEN
    //-------------------------------------
    StepCompleteWhen(Station.UpdateEntityTask.Done);
    //-------------------------------------	
END_IF


//monitor if conseccutive failures occur during automatic cycle. System monitor two basic types like are arbitrary failure in seqence, or  same(equal) failure in sequence
//if Number of allowed recurring failure is 0 , monitoring is inactive.
//Recurring failures are based on ErrorCodes in TcoComprehensiveResult.
//If error code in Same recurring failure is empty string ,monitorig of failure is not performed.
//Error code in Arbitrary Recuring failure is irelevant.    
THIS^.MonitorAnyRecurringFailure(22000,THIS^.Station._settings.AnyRecurringFailure>0 , Station.ProcessDataManager.Data.EntityHeader.Results);
THIS^.MonitorSameRecurringFailure(22100,THIS^.Station._settings.SameRecurringFailure>0 , Station.ProcessDataManager.Data.EntityHeader.Results);



IF (Step(30000, TRUE, 'LAST STEP')) THEN
    //-------------------------------------
    IF (_loop) THEN
        CompleteSequence();
    END_IF;
    //-------------------------------------	
END_IF

_paralellTask();
END_METHOD

METHOD PUBLIC OnStart
SUPER^.OnStart();
Station.GroundTask.Restore();
Station.ManualTask.Restore();
Station.GroundTask.CancelGround();
_paralellTask.Restore();
END_METHOD

METHOD SingleExample : BOOL
VAR_INPUT
		inStepID : INT;
END_VAR

IF (Step(inStepID, TRUE, 'SINGLE INSPECTION')) THEN
    //-------------------------------------    
	Station.ProcessDataManager.Data.CU00x.BoltPresenceInspector.Data.FailureDescription:='BoltPresenceInspector error';
    Station.ProcessDataManager.Data.CU00x.BoltPresenceInspector.WithCoordinator(THIS^)
        .Inspect(_inspectionResult)
        .UpdateComprehensiveResult(Station.ProcessDataManager.Data.EntityHeader.Results)
        .OnFail().Dialog(inStepID+10);
    //-------------------------------------
END_IF

// with checking if specific inspector is overinspected
IF (Step(inStepID+10, TRUE, 'SINGLE ANALOGUE INSPECTION')) THEN
//-------------------------------------
	Station.ProcessDataManager.Data.CU00x.BoltDimensionPresenceInspector.Data.FailureDescription:='BoltDimensionPresenceInspector error';
	Station.ProcessDataManager.Data.CU00x.BoltDimensionPresenceInspector.Data.NumberOfAllowedRetries:=100;
	IF NOT Station.ProcessDataManager.Data.CU00x.BoltDimensionPresenceInspector.OverInspected THEN
	
		Station.ProcessDataManager.Data.CU00x.BoltDimensionPresenceInspector.WithCoordinator(THIS^)
			.Inspect(_inspectionDimensionResult)
			.WithDescription()
			.UpdateComprehensiveResult(Station.ProcessDataManager.Data.EntityHeader.Results)
			.OnFail().Retry(inStepID+20);
	ELSE
	 	RequestStep(RESTORE_STEP_ID);	
	END_IF
//-------------------------------------
END_IF;

IF (Step(inStepID+20, TRUE, 'DONE')) THEN
//-------------------------------------
		CompleteStep();
//-------------------------------------
END_IF;
END_METHOD

PROPERTY Station : REFERENCE TO CU00x
GET
VAR
    _station : POINTER TO CU00x;
END_VAR
IF __QUERYPOINTER(Parent, _station) THEN // Check if _Parent is Station001
    Station REF= _station^;              // If the check is successful dereference a pointer. simlar to THIS^ or SUPER^
END_IF
END_GET
END_PROPERTY

END_FUNCTION_BLOCK

// ---- Technology/CU00x/Automat/CU00xAutomatParalell_1_Task.TcPOU
FUNCTION_BLOCK CU00xAutomatParalell_1_Task EXTENDS TcoTaskedSequencer 

VAR
	_customTimer: TON;
END_VAR

Run();

(*~
	<docu>
		<summary>
			Main method of the sequener. Custom code needs to be placed here. The sequencer is executed by call of **Instance.Run()** method.
			This method is abstract, and it must be overridden in derived block.
		</summary>
	</docu>
~*)
METHOD PROTECTED Main : BOOL
// Takes mode (step/continous) from the parent controller
THIS^.ModeController.Mode := ParentSequence.ModeController.Mode;

IF (Step(1000, TRUE, 'PARALELL STEP - EXAMPLE OF TIMERS')) THEN
    //-------------------------------------    
		StepCompleteWhen(CurrentStep.Duration >= T#300mS);	
    //-------------------------------------
END_IF
IF (Step(1100, TRUE, 'PARALELL STEP - EXAMPLE OF TIMERS')) THEN
    //-------------------------------------    
		StepCompleteWhen(inCondition:=Timer_1(TRUE,T#100MS));	
    //-------------------------------------
END_IF
IF (Step(1200, TRUE, 'PARALELL STEP - EXAMPLE OF TIMERS')) THEN
    //-------------------------------------    
		StepCompleteWhen(inCondition:=Timer_1(TRUE,T#200MS));	
    //-------------------------------------
END_IF

IF THIS^.IsFreshState THEN
	_customTimer(IN:=FALSE);
END_IF
IF (Step(1300, TRUE, 'PARALELL STEP - EXAMPLE OF TIMERS')) THEN
    //-------------------------------------    

		_customTimer(IN:=TRUE,PT:=T#200MS);
		StepCompleteWhen(inCondition:=_customTimer.Q);	
    //-------------------------------------
END_IF


IF (Step(10000, TRUE, 'PARALELL TASK DONE')) THEN
    //-------------------------------------
    _task.DoneWhen(TRUE );
    //-------------------------------------	
END_IF
END_METHOD

PROPERTY ParentSequence : REFERENCE TO CU00xAutomatTask
GET
VAR
    _parentSequence : POINTER TO CU00xAutomatTask;
END_VAR
IF __QUERYPOINTER(Parent, _parentSequence) THEN 
    ParentSequence REF= _parentSequence^;              
END_IF
END_GET
END_PROPERTY

END_FUNCTION_BLOCK

// ---- Technology/CU00x/Data/CU00xDialogContent.TcPOU
FUNCTION_BLOCK CU00xDialogContent EXTENDS TcoCore.TcoInputDialogContentContainer
VAR_INPUT
END_VAR
VAR_OUTPUT
END_VAR
VAR
	{attribute addProperty Name "<#Recipe#>"}
	Recipe:STRING;
	{attribute addProperty Name "<#Qantity#>"}
	RequiredQuantity:INT;
	{attribute addProperty Name "<#Timeout#>"}
	Timeout:DATE_AND_TIME;
	{attribute addProperty Name "<#Exclude#>"}
	Exclude:BOOL;

END_VAR

END_FUNCTION_BLOCK

// ---- Technology/CU00x/Safety/Suspend/CU00xSuspendTask.TcPOU
FUNCTION_BLOCK CU00xSuspendTask EXTENDS CUBaseSuspend IMPLEMENTS ICUTask
VAR
	_sb : TcoCore.StringBuilder;
END_VAR

Run();

(*~
	<docu>
		<summary>
			Main method of the sequener. Custom code needs to be placed here. The sequencer is executed by call of **Instance.Run()** method.
			This method is abstract, and it must be overridden in derived block.
		</summary>
	</docu>
~*)
METHOD PROTECTED Main : BOOL
(*

	SUSPEND PROCESS 
	Following steps provide suspend actions for this controlled unit.
	Add components add write customized sequence according to your need.
*)

		
//
IF (Step(100, TRUE, '<#WAITING FOR START#>')) THEN
    //-------------------------------------    

    StepCompleteWhen(TRUE);
    //-------------------------------------
END_IF

//HERE  YOU CAN WRITE  WHAT IS NECESSARY 
//TO SUPSEND  PROCESS..... TO INTERUPT SAFETY

IF (Step(1000, TRUE, '<#SUSPENDING COMPONENTS#>')) THEN
 	//-------------------------------------    
	//StepCompleteWhen(Station.AutomatTask.CurrentStep.Status <> eStepStatus.Running);
		
    StepCompleteWhen( CurrentStep.Duration >= T#3000MS);
    //-------------------------------------
END_IF

IF (Step(30000, TRUE, 'SUSPEND DONE')) THEN
    //-------------------------------------
		
        THIS^._done:=TRUE;
		THIS^.Task.DoneWhen(TRUE);
	
   
    //-------------------------------------	
END_IF
END_METHOD

METHOD PUBLIC OnStart
SUPER^.OnStart();
Station.RecoverTask.Restore();
END_METHOD

PROPERTY Station : REFERENCE TO CU00x
GET
VAR
    _station : POINTER TO CU00x;
END_VAR
IF __QUERYPOINTER(Parent, _station) THEN // Check if _Parent is Station001
    Station REF= _station^;              // If the check is successful dereference a pointer. simlar to THIS^ or SUPER^
END_IF
END_GET
END_PROPERTY

END_FUNCTION_BLOCK

// ---- Technology/CU00x/Safety/Recover/CU00xRecoverTask.TcPOU
FUNCTION_BLOCK CU00xRecoverTask EXTENDS CUBaseRecover IMPLEMENTS ICUTask
VAR
	_sb : TcoCore.StringBuilder;
END_VAR

Run();

(*~
	<docu>
		<summary>
			Main method of the sequener. Custom code needs to be placed here. The sequencer is executed by call of **Instance.Run()** method.
			This method is abstract, and it must be overridden in derived block.
		</summary>
	</docu>
~*)
METHOD PROTECTED Main : BOOL
(*

	RECOVER PROCESS 
	Following steps provide recover action for this controlled unit.
	Add components add write customized sequence according to your need.
*)

		
//
IF (Step(100, TRUE, '<#WAITING FOR START#>')) THEN
    //-------------------------------------    

    StepCompleteWhen(TRUE);
    //-------------------------------------
END_IF

//HERE  YOU CAN WRITE  WHAT IS NECESSARY 
//TO RECOVER AFTER INTERUPTED PROCESS.....

IF (Step(1000, TRUE, '<#RECOVER ANY COMPONENTS#>')) THEN
    //-------------------------------------    

    StepCompleteWhen(CurrentStep.Duration >= T#3000MS);
    //-------------------------------------
END_IF

IF (Step(30000, TRUE, 'RECOVER DONE')) THEN
    //-------------------------------------
		
        this^._done:=true;
		THIS^.Task.DoneWhen(TRUE);
		
   
    //-------------------------------------	
END_IF
END_METHOD

METHOD PUBLIC OnStart
SUPER^.OnStart();
Station.SuspendTask.Restore();
END_METHOD

PROPERTY Station : REFERENCE TO CU00x
GET
VAR
    _station : POINTER TO CU00x;
END_VAR
IF __QUERYPOINTER(Parent, _station) THEN // Check if _Parent is Station001
    Station REF= _station^;              // If the check is successful dereference a pointer. simlar to THIS^ or SUPER^
END_IF
END_GET
END_PROPERTY

END_FUNCTION_BLOCK

// ---- Technology/CU00x/Positions/Cu00xTestPositions.TcPOU
FUNCTION_BLOCK Cu00xTestPositions EXTENDS TcoDrivesBeckhoff.TcoSingleAxisPositionsRootContainer
VAR_INPUT
END_VAR
VAR_OUTPUT
END_VAR
VAR
	{attribute addProperty Name "<#Pick Position#>"}
	PickPosition:TcoDrivesBeckhoff.TcoSingleAxisMoveParam;
	{attribute addProperty Name "<#Place  Position#>"}
	PlacePosition:TcoDrivesBeckhoff.TcoSingleAxisMoveParam;
END_VAR

END_FUNCTION_BLOCK

// ---- Technology/CU00x/Positions/CU00xTestMultiPositions.TcPOU
FUNCTION_BLOCK CU00xTestMultiPositions EXTENDS TcoDrivesBeckhoff.TcoMultiAxisPositionsRootContainer
VAR_INPUT
END_VAR
VAR_OUTPUT
END_VAR
VAR
	{attribute addProperty Name "<#Pick Position#>"}
	PickPosition:TcoDrivesBeckhoff.TcoMultiAxisMoveParam;
	{attribute addProperty Name "<#Place  Position#>"}
	PlacePosition:TcoDrivesBeckhoff.TcoMultiAxisMoveParam;

END_VAR

PROPERTY PUBLIC PickPos : REFERENCE TO TcoDrivesBeckhoff.TcoMultiAxisMoveParam;
GET
PickPos REF=PickPosition;
END_GET
END_PROPERTY

PROPERTY PUBLIC PlacePos : REFERENCE TO TcoDrivesBeckhoff.TcoMultiAxisMoveParam;
GET
PlacePos REF=PlacePosition;
END_GET
END_PROPERTY

END_FUNCTION_BLOCK

// ---- Abstractions/Components/MtsFeeding/TcoFeedingSequenceTask.TcPOU
FUNCTION_BLOCK TcoFeedingSequenceTask EXTENDS TcoCore.TcoTask
VAR
	_sequence      : TcoCore.TcoSequence(THIS^, eRestoreMode.None);
    _observerSequence       : TcoCore.TcoSequencerObserver(THIS^);
END_VAR

PROPERTY PUBLIC Observer : REFERENCE TO TcoCore.TcoSequencerObserver
GET
Observer ref=_observerSequence;
END_GET
END_PROPERTY

(*~
	<docu>
		<summary>
			Restores this instance to the Ready state. Can be called explicitly or from within one of the restore mechanisms.
			<para>
				See also <see cref="PlcDocu.TcoCore.TcoTask.AutoRestorable()"/>
			</para>
		</summary>			
	</docu>	
~*)
METHOD Restore : ITcoRestorable
SUPER^.Restore();
_sequence.Restore();
END_METHOD

PROPERTY PUBLIC Sequence : REFERENCE TO TcoCore.TcoSequence
GET
Sequence ref=_sequence;
END_GET
END_PROPERTY

END_FUNCTION_BLOCK

// ---- Abstractions/Components/MtsFeeding/TcoPlsPaletizator.TcPOU
FUNCTION_BLOCK TcoPlsPaletizator EXTENDS TcoCore.TcoComponent
VAR_INPUT
	inSafeCondition:BOOL;
	inDoorOpen:BOOL;
END_VAR

VAR_OUTPUT
END_VAR
VAR
	 {attribute addProperty Name "<#Config#>"}
	_config:TcoPlsPaletizator_Config_v_1_x_x;
	 {attribute addProperty Name "<#Status#>"}
    {attribute clr [ReadOnly()]}
	_status:TcoPlsPaletizator_Status_v_1_x_x;
	 {attribute addProperty Name "<#Control#>"}
	_control:TcoPlsPaletizator_Control_v_1_x_x;
	
	 {attribute addProperty Name "<#Components#>"}
    _components:TcoPlsPaletizator_Components:= (Parent := THIS^);
	
	{attribute addProperty Name "<#Poziadavka novy blister#>"}
	_feedNewBlisterTask : TcoFeedingSequenceTask(THIS^);
	{attribute addProperty Name "<#Poziadavka vylozenie blistera#>"}
	_throwBlisterTask :  TcoFeedingSequenceTask(THIS^);
	{attribute addProperty Name "<#Poziadavka obsluhy vystupny buffer#>"}
	_hanldeOutBufferTask :  TcoFeedingSequenceTask(THIS^);


	
	{attribute addProperty Name "<#Restore#>"}
	_restoreTask:TcoCore.TcoTask(THIS^);

	_blinker:TcoBlinker(THIS^);
	restoreDone: BOOL;
END_VAR

_status.SafeCondition:=inSafeCondition;
_status.EntryBufferEmpty:=NOT Components.I3_PresentBlistersInBufferEmpty.Signal;
_status.BlisterReady:= Components.I4_PresentBlisterInWorkingPos.Signal ;
_status.OutBufferFull:= Components.I8_OutBlistersBufferIsFull.Signal;

_feedNewBlisterTask.Enabled :=NOT _throwBlisterTask.Busy;
IF(_feedNewBlisterTask.Execute())THEN
	SequenceIncomingBlister(refSequenceTask:=_feedNewBlisterTask );
END_IF;

_throwBlisterTask.Enabled :=NOT _feedNewBlisterTask.Busy;
IF(_throwBlisterTask.Execute())THEN
	SequenceOutgoingBlister(refSequenceTask:=_throwBlisterTask);
END_IF;

_hanldeOutBufferTask.Enabled :=TRUE;
IF(_hanldeOutBufferTask.Execute())THEN
	SequenceOutgoingBuffer(refSequenceTask:=_hanldeOutBufferTask);
END_IF;



//*************RESTORE********************

_restoreTask.Enabled := TRUE;
IF _restoreTask.Execute() THEN
	Restore();
	restoreDone:= Components.P3_HorizontalSepareEntryBlisters.MoveToWork().Done AND (Components.P10_HoldEntrySepareOutBlister.MoveToHome().Done or _config.SepareBlistersAtEntryInactive)
		AND_THEN (Components.P1_VerticalSepareEntryBlisters.MoveToHome().Done AND Components.P2_VerticalSepareEntryBlisters.MoveToHome().Done)
		AND_THEN (Components.P5_HorizontalSepareOutBlisters.MoveToHome().Done AND_THEN Components.P6_VerticalSepareOutBlister.MoveToHome().Done)
		AND_THEN  Components.P4_FeedEntryBlister.MoveToHome().Done;
		
	
	_restoreTask.DoneWhen(restoreDone);
END_IF
//****************************************

PROPERTY Components : REFERENCE TO TcoPlsPaletizator_Components
GET
Components ref=_components;
END_GET
END_PROPERTY

(*~
	<docu>
		<summary>
			Gets the configuration of the MTS Pls feeder. 					
		</summary>			
	</docu>	
~*)
PROPERTY Config : REFERENCE TO TcoPlsPaletizator_Config_v_1_x_x
GET
Config REF= _config;
END_GET
END_PROPERTY

METHOD PUBLIC DefaultSignalisation
VAR_INPUT
END_VAR
Components.Q1_AttentionSignalisationR.Reset();
Components.Q2_AttentionSignalisationG.Reset();
Components.Q3_AttentionSignalisationB.Reset();

_blinker(inOffTime:=_config.BlinkTime,inOnTime:=_config.BlinkTime);

IF NOT _status.OutBufferFull 
	AND NOT _status.EntryBufferEmpty THEN
	Components.Q2_AttentionSignalisationG.Set();
ELSIF  _blinker.IsOn THEN
	IF inDoorOpen AND 
		THIS^._feedNewBlisterTask.Busy
		OR
		THIS^._throwBlisterTask.Busy
		OR
		THIS^._hanldeOutBufferTask.Busy THEN
		Messenger.Warning('<#CAKANIE NA OBSLUHU PALETIZERA - ZAVRITE DVERE!#>');
		Components.Q1_AttentionSignalisationR.Set();
		Components.Q2_AttentionSignalisationG.Set();
	ELSIF NOT _status.OutBufferFull
		AND _status.EntryBufferEmpty
		AND _status.BlisterReady THEN
		
		Components.Q1_AttentionSignalisationR.Set();
		Components.Q2_AttentionSignalisationG.Set();

	ELSIF NOT _status.OutBufferFull
		AND _status.EntryBufferEmpty 
		AND NOT _status.BlisterReady THEN	
		Components.Q1_AttentionSignalisationR.Set();
	ELSIF  _status.OutBufferFull  THEN
		Components.Q1_AttentionSignalisationR.Set();	
	
	END_IF;


	
END_IF;
END_METHOD

PROPERTY FeedNewBlisterTask : REFERENCE TO TcoFeedingSequenceTask
GET
FeedNewBlisterTask ref=_feedNewBlisterTask;
END_GET
END_PROPERTY

PROPERTY HandleOutBufferTask : REFERENCE TO TcoFeedingSequenceTask
GET
HandleOutBufferTask ref=_hanldeOutBufferTask;
END_GET
END_PROPERTY

(*~
	<docu>
		<summary>
			Restores this instance to the Ready state. Can be called explicitly or from within one of the restore mechanisms.	
		</summary>			
	</docu>	
~*)
METHOD  Restore : ITcoRestorable

_hanldeOutBufferTask.Restore();
_feedNewBlisterTask.Restore();
_throwBlisterTask.Restore();
END_METHOD

METHOD PUBLIC SafetyBlockingMovements
VAR_INPUT
END_VAR
//********************SAFETY******************

Components.P4_FeedEntryBlister.SuspendMoveWorkExpression(NOT Components.P7_SupportEntryBlister.AtHome ,'Movement is blocked due P7 is not in home position');
Components.P4_FeedEntryBlister.SuspendMoveHomeExpression(NOT Components.P6_VerticalSepareOutBlister.AtHome,'Movement is blocked due P6 is not in home position');
END_METHOD

METHOD SequenceIncomingBlister
VAR_INPUT
	refSequenceTask : REFERENCE TO TcoFeedingSequenceTask;
	
	
END_VAR

VAR
    seq    : REFERENCE TO TcoCore.TcoSequence;


END_VAR
seq REF= refSequenceTask.Sequence;

seq.Open();
seq.Observer := refSequenceTask.Observer;



		



//***************************************************************************************************     
//    This step will be executed and immediately finished, as the condition in Await method is true.
IF seq.Step(0,TRUE,'<#INIT#>') THEN   
	Messenger.Warning('<#BEZPECNOST ZARIADENIA NARUSENA. NIEJE MOZNE VYKONAT AKCIU#>');     
	IF _status.SafeCondition THEN
    	seq.CompleteStep();
	END_IF;
END_IF        
//***************************************************************************************************     

 
//***************************************************************************************************     
IF seq.Step(10,TRUE,'<#KONTROLA POCTU VSTUPNYCH BLISTROV#>') THEN   
    Messenger.Warning('<#PODAVAC PRAZDNY! DOPLNE VSTUPNE BLISTRE !#>');
    seq.StepCompleteWhen(Components.I3_PresentBlistersInBufferEmpty.IsTrue);
END_IF        
//***************************************************************************************************     


        
//***************************************************************************************************     
IF seq.Step(20,TRUE,'<#SEPAROVANIE VSTUPNEHO BLISTRA - VERTIKALNE VALCE VYSUNUTE#>') THEN   

    seq.StepCompleteWhen(THIS^.Components.P1_VerticalSepareEntryBlisters.MoveToWork().Done AND THIS^.Components.P2_VerticalSepareEntryBlisters.MoveToWork().Done);
END_IF        
//***************************************************************************************************     


//***************************************************************************************************     
IF seq.Step(30,TRUE,'<#SEPAROVANIE VSTUPNEHO BLISTRA - SEPAROVANIE ZASUNUTE#>') THEN   

    seq.StepCompleteWhen(THIS^.Components.P3_HorizontalSepareEntryBlisters.MoveToHome().Done);
END_IF        
//***************************************************************************************************     


//***************************************************************************************************     
IF seq.Step(40,TRUE,'<#SEPAROVANIE VSTUPNEHO BLISTRA - VERTIKALNE VALCE ZASUNUT JEDEN#>') THEN   

    seq.StepCompleteWhen(THIS^.Components.P1_VerticalSepareEntryBlisters.MoveToHome().Done AND_THEN THIS^.Components.P2_VerticalSepareEntryBlisters.MoveToWork().Done);
END_IF        
//***************************************************************************************************     


//***************************************************************************************************     
IF seq.Step(50,TRUE,'<#SEPAROVANIE VSTUPNEHO BLISTRA - SEPAROVANIE VYSUNUTE#>') THEN   

    seq.StepCompleteWhen(THIS^.Components.P3_HorizontalSepareEntryBlisters.MoveToWork().Done AND (Components.P10_HoldEntrySepareOutBlister.MoveToWork().Done or _config.SepareBlistersAtEntryInactive));
END_IF        
//***************************************************************************************************     

//***************************************************************************************************     
IF seq.Step(60,TRUE,'<#SEPAROVANIE VSTUPNEHO BLISTRA - VERTIKALNE VALCE ZASUNUT OBIDVA#>') THEN   

    seq.StepCompleteWhen(THIS^.Components.P1_VerticalSepareEntryBlisters.MoveToHome().Done AND THIS^.Components.P2_VerticalSepareEntryBlisters.MoveToHome().Done 
						AND_THEN (Components.P10_HoldEntrySepareOutBlister.MoveToHome().Done) OR _config.SepareBlistersAtEntryInactive);
END_IF        
//***************************************************************************************************     

//***************************************************************************************************   
IF seq.Step(70,TRUE,'<#KONTROLA PRITOMNOSTI SEPAROVANEHO KUSU#>') THEN   
    Messenger.Error('<#PODAVAC PRAZDNY! DOPLNE BLISTRE !#>');
    seq.StepCompleteWhen(THIS^.Components.I1_PresentBlisterEntry.IsTrue AND (THIS^.Components.I2_PresentBlisterEntryEmptySpace.IsTrue) );
END_IF        
//***************************************************************************************************     


//***************************************************************************************************     
IF seq.Step(80,TRUE,'<#SEPAROVANIE VSTUPNEHO BLISTRA - PRESUNUTIE BLISTRA DO POZICIE ODOBERANIA#>') THEN   

    seq.StepCompleteWhen(THIS^.Components.P8_FixEntryBlisterSide.MoveToHome().Done AND_THEN THIS^.Components.P4_FeedEntryBlister.MoveToWork().Done AND Components.i4_PresentBlisterInWorkingPos.IsTrue);
END_IF        
//***************************************************************************************************     


//***************************************************************************************************     
IF seq.Step(90,TRUE,'<#SEPAROVANIE VSTUPNEHO BLISTRA - UPEVENIE BLISTRA ZBOKU#>') THEN   

    seq.StepCompleteWhen(THIS^.Components.P8_FixEntryBlisterSide.MoveToWork().Done);
END_IF        
//***************************************************************************************************     



//***************************************************************************************************     
IF seq.Step(100,TRUE,'<#SEPAROVANIE VSTUPNEHO BLISTRA - NPRESUNUTIE BLISTRA DO POZICIE NABERANIA#>') THEN   

   IF THIS^.Components.P6_VerticalSepareOutBlister.AtHome THEN
	    seq.CompleteStep();
	ELSE
		Messenger.Error('VYSTUPNY BUFFER NIEJE V HORNEJ POZICII!(P6)');
	END_IF
END_IF        
//***************************************************************************************************   

//***************************************************************************************************     
IF seq.Step(110,TRUE,'<#SEPAROVANIE VSTUPNEHO BLISTRA - ZASUNUTE P4#>') THEN   

	 seq.StepCompleteWhen(THIS^.Components.P4_FeedEntryBlister.MoveToHome().Done) ;
	
END_IF        
//***************************************************************************************************   


//***************************************************************************************************     
IF seq.Step(120,TRUE,'SEPAROVANIE VSTUPNEHO BLISTRA - NPRESUNUTIE BLISTRA DO POZICIE NABERANIA') THEN   

    seq.StepCompleteWhen(THIS^.Components.P7_SupportEntryBlister.MoveToWork().Done AND (THIS^.Components.P9_LockEntryBlisterTop.MoveToHome().Done OR _config.LockBlisterInPickPosInactive));
END_IF        
//***************************************************************************************************   




IF (seq.Step(inStepID := seq.RESTORE_STEP_ID,
    inEnabled := TRUE,
    inStepDescription := 'RETURN TO THE START OF THE SEQUENCE')) THEN
    //--------------------------------------------------------	
		refSequenceTask.DoneWhen(TRUE);
    	seq.CompleteSequence();
    //--------------------------------------------------------			
END_IF;

seq.Close();
END_METHOD

METHOD SequenceOutgoingBlister
VAR_INPUT
	refSequenceTask : REFERENCE TO TcoFeedingSequenceTask;
	
	
END_VAR

VAR
    seq    : REFERENCE TO TcoCore.TcoSequence;

END_VAR

VAR_INST
	_timer:ton;
	
END_VAR
seq REF= refSequenceTask.Sequence;

seq.Open();
seq.Observer := refSequenceTask.Observer;



		



//***************************************************************************************************     
//    This step will be executed and immediately finished, as the condition in Await method is true.
IF seq.Step(0,TRUE,'<#INIT#>') THEN   
	Messenger.Warning('<#BEZPECNOST ZARIADENIA NARUSENA. NIEJE MOZNE VYKONAT AKCIU#>');     
	IF _status.SafeCondition THEN
    	seq.CompleteStep();
	END_IF;
END_IF        
//***************************************************************************************************     

IF seq.Step(10,TRUE,'<#SEPAROVANIE VYSTUPNEHO BLISTRA - UVOLNENIE BLISTRA#>') THEN   

    seq.StepCompleteWhen( (THIS^.Components.P9_LockEntryBlisterTop.MoveToWork().Done OR _config.LockBlisterInPickPosInactive) AND THIS^.Components.P8_FixEntryBlisterSide.MoveToHome().Done);
END_IF        
//***************************************************************************************************   


//***************************************************************************************************     
IF seq.Step(20,TRUE,'<#SEPAROVANIE VYSTUPNEHO BLISTRA - ZASUNUTIE SUPPORTU#>') THEN   

   seq.StepCompleteWhen(THIS^.Components.P7_SupportEntryBlister.MoveToHome().Done);
END_IF        
//***************************************************************************************************   



//***************************************************************************************************     
IF seq.Step(30,TRUE,'<#SEPAROVANIE VYSTUPNEHO BLISTRA - KONTROLA PRITOMNOSTI BLISTA NA SKLZE#>') THEN   
	IF seq.IsFreshState THEN
		_timer(IN:=FALSE);
	END_IF
	_timer(IN:=THIS^.Components.I5_OutBlistersIsThrowedCorrectly.Signal,PT:=_config.StabilisationTime);
	
    seq.StepCompleteWhen(_timer.Q);
END_IF        
//***************************************************************************************************   



IF (seq.Step(inStepID := seq.RESTORE_STEP_ID,
    inEnabled := TRUE,
    inStepDescription := 'RETURN TO THE START OF THE SEQUENCE')) THEN
    //--------------------------------------------------------	
		refSequenceTask.DoneWhen(TRUE);
    	seq.CompleteSequence();
    //--------------------------------------------------------			
END_IF;

seq.Close();
END_METHOD

METHOD SequenceOutgoingBuffer
VAR_INPUT
	refSequenceTask : REFERENCE TO TcoFeedingSequenceTask;
	
	
END_VAR

VAR
    seq    : REFERENCE TO TcoCore.TcoSequence;

END_VAR

VAR_INST
	_timer:ton;
	
END_VAR
seq REF= refSequenceTask.Sequence;

seq.Open();
seq.Observer := refSequenceTask.Observer;



		



//***************************************************************************************************     
//    This step will be executed and immediately finished, as the condition in Await method is true.
IF seq.Step(0,TRUE,'<#INIT#>') THEN   
	Messenger.Warning('<#BEZPECNOST ZARIADENIA NARUSENA. NIEJE MOZNE VYKONAT AKCIU#>');     
	IF _status.SafeCondition THEN
    	seq.CompleteStep();
	END_IF;
END_IF        
//***************************************************************************************************     



//***************************************************************************************************     
IF seq.Step(10,TRUE,'<#VYSTUPNY BUFFER - KONTROLA PRITOMNOSTI BLISTA NAD BUFFEROM#>') THEN   
	IF seq.IsFreshState THEN
		_timer(IN:=FALSE);
	END_IF
	_timer(IN:=NOT THIS^.Components.I5_OutBlistersIsThrowedCorrectly.Signal AND Components.I7_OutBlistersIsAboveOutBuffer.Signal,PT:=_config.StabilisationTime);
	
    seq.StepCompleteWhen(_timer.Q);
END_IF        
//***************************************************************************************************   


//***************************************************************************************************     
IF seq.Step(20,TRUE,'<#VYSTUPNY BUFFER - KONTROLA POSCTU BLISTROV#>') THEN   
	Messenger.Error('<#PODAVAC PLNY! ODSTRANTE PRAZDNE BLISTRE !#>');
    seq.StepCompleteWhen(THIS^.Components.I8_OutBlistersBufferIsFull.IsFalse);
END_IF        
//***************************************************************************************************   


//***************************************************************************************************     
IF seq.Step(30,TRUE,'<#VYSTUPNY BUFFER - POSUN KUSOV NAD BUFFER#>') THEN   

	THIS^.Components.P6_VerticalSepareOutBlister.MoveToWork();
	IF Components.I6_OutBlistersLisftSignal.Signal THEN
	
		THIS^.Components.P6_VerticalSepareOutBlister.MoveWorkTask.Abort();
	    seq.StepCompleteWhen(TRUE);
	END_IF;
		
END_IF        
//***************************************************************************************************   


//***************************************************************************************************     
IF seq.Step(40,TRUE,'<#VYSTUPNY BUFFER - UVOLNENIE BLISTRA A NAVRAT NAHOR#>') THEN   

	
	seq.StepCompleteWhen(Components.P5_HorizontalSepareOutBlisters.MoveToWork().Done AND_THEN THIS^.Components.P6_VerticalSepareOutBlister.MoveToHome().Done);
		
END_IF        
//***************************************************************************************************   

//***************************************************************************************************     
IF seq.Step(50,TRUE,'<#VYSTUPNY BUFFER - HORIZONTALNE ZASUNUTIE#>') THEN   

	
	seq.StepCompleteWhen(Components.P5_HorizontalSepareOutBlisters.MoveToHome().Done);
		
END_IF        
//***************************************************************************************************   



IF (seq.Step(inStepID := seq.RESTORE_STEP_ID,
    inEnabled := TRUE,
    inStepDescription := 'RETURN TO THE START OF THE SEQUENCE')) THEN
    //--------------------------------------------------------	
		refSequenceTask.DoneWhen(TRUE);
    	seq.CompleteSequence();
    //--------------------------------------------------------			
END_IF;

seq.Close();
END_METHOD

(*~
	<docu>
		<summary>
		    Custom service (manual, maintenance) logic.
			This method must be implemented in derived class.
		</summary>			
	</docu>	
~*)
METHOD PROTECTED  ServiceMode
_components.Q3_AttentionSignalisationB.Service();
_components.Q2_AttentionSignalisationG.Service();
_components.Q1_AttentionSignalisationR.Service();
_components.P1_VerticalSepareEntryBlisters.Service();
_components.P2_VerticalSepareEntryBlisters.Service();
_components.P3_HorizontalSepareEntryBlisters.Service();
_components.P4_FeedEntryBlister.Service();
_components.P5_HorizontalSepareOutBlisters.Service();
_components.P6_VerticalSepareOutBlister.Service();
_components.P7_SupportEntryBlister.Service();
_components.P8_FixEntryBlisterSide.Service();
_components.P9_LockEntryBlisterTop.Service();
_components.P10_HoldEntrySepareOutBlister.Service();
END_METHOD

(*~
	<docu>
		<summary>
			Gets the status of the MTS Pls feeder. 					
		</summary>			
	</docu>	
~*)
PROPERTY Status : REFERENCE TO TcoPlsPaletizator_Status_v_1_x_x
GET
Status REF= _status;
END_GET
END_PROPERTY

PROPERTY ThrowBlisterTask : REFERENCE TO TcoFeedingSequenceTask
GET
ThrowBlisterTask ref=_throwBlisterTask;
END_GET
END_PROPERTY

END_FUNCTION_BLOCK

// ---- Abstractions/Components/WrappedComponent/WrappedComponentExample.TcPOU
FUNCTION_BLOCK WrappedComponentExample EXTENDS TcoCore.TcoComponent


VAR_OUTPUT
END_VAR
VAR
	_config:WrappedComponentExample_Config;
	_status:WrappedComponentExample_Status;
	_control:WrappedComponentExample_Control;
    _components:WrappedComponentsExample:= (Parent := THIS^);
	_throwTask:TcoCore.TcoTask(THIS^);
	_restoreTask:TcoCore.TcoTask(THIS^);

END_VAR

_throwTask();
_restoreTask.Enabled:=true;
_restoreTask();

PROPERTY Components : REFERENCE TO WrappedComponentsExample
GET
Components ref=_components;
END_GET
END_PROPERTY

(*~
	<docu>
		<summary>
			Restores this instance to the Ready state. Can be called explicitly or from within one of the restore mechanisms.	
		</summary>			
	</docu>	
~*)
METHOD  Restore : ITcoRestorable
END_METHOD

(*~
	<docu>
		<summary>
		    Custom service (manual, maintenance) logic.
			This method must be implemented in derived class.
		</summary>			
	</docu>	
~*)
METHOD PROTECTED  ServiceMode
END_METHOD

END_FUNCTION_BLOCK

// ---- Abstractions/Safety/ControlButtons/TcoControlButtons.TcPOU
{attribute wpf [Container(Layout.Stack)]}
FUNCTION_BLOCK TcoControlButtons EXTENDS TcoCore.TcoObject IMPLEMENTS ITcoControlButtons
VAR_IN_OUT
    {attribute clr [RenderIgnore()]}
    inoButtonRecover : bool;
    {attribute clr [RenderIgnore()]}
    inoButtonSuspend : BOOL;
	{attribute clr [RenderIgnore()]}
    inoButtonGround : BOOL;
    {attribute clr [RenderIgnore()]}
    inoButtonAuto : BOOL;
    {attribute clr [RenderIgnore()]}
    inoButtonRecoverLight : BOOL;
    {attribute clr [RenderIgnore()]}
    inoButtonSuspendLight : BOOL;
    {attribute clr [RenderIgnore()]}
    inoButtonGroundLight : BOOL;
    {attribute clr [RenderIgnore()]}
    inoButtonAutoLight : BOOL;

END_VAR
VAR


    {attribute addProperty Name "<#ButtonRecover#>"}
    _buttonRecover : TcoElements.TcoDi(THIS^);

    {attribute addProperty Name "<#ButtonSuspend#>"}
    _buttonSuspend : TcoElements.TcoDi(THIS^);

    {attribute addProperty Name "<#ButtonGround#>"}
    _buttonGround : TcoElements.TcoDi(THIS^);

    {attribute addProperty Name "<#ButtonAuto#>"}
    _buttonAuto : TcoElements.TcoDi(THIS^);



    {attribute addProperty Name "<#ButtonStartLight#>"}
    _buttonRecoverLight : TcoElements.TcoDo(THIS^);

    {attribute addProperty Name "<#ButtonStopLight#>"}
    _buttonSuspendLight : TcoElements.TcoDo(THIS^);

    {attribute addProperty Name "<#ButtonGroundLight#>"}
    _buttonGroundLight : TcoElements.TcoDo(THIS^);
    {attribute addProperty Name "<#ButtonAutoLight#>"}
    _buttonAutoLight : TcoElements.TcoDo(THIS^);


END_VAR

_buttonRecover(inoSignal:= inoButtonRecover);
_buttonSuspend(inoSignal:= inoButtonSuspend);
_buttonGround(inoSignal:= inoButtonGround);
_buttonAuto(inoSignal:= inoButtonAuto);



_buttonGroundLight(inoSignal:= inoButtonGroundLight);
_buttonSuspendLight(inoSignal:= inoButtonSuspendLight);
_buttonRecoverLight(inoSignal:= inoButtonRecoverLight);
_buttonAutoLight(inoSignal:= inoButtonAutoLight);

PROPERTY ButtonAuto : BOOL
GET
ButtonAuto :=  _buttonAuto._signal;
END_GET
SET
// Light up illumination of button
IF ButtonAuto THEN
	_buttonAutoLight.Set();
ELSE
	_buttonAutoLight.Reset();
END_IF
END_SET
END_PROPERTY

PROPERTY ButtonGround : BOOL
GET
ButtonGround :=  _buttonGround._signal;
END_GET
SET
// Light up illumination of button
IF ButtonGround THEN
	_buttonGroundLight.Set();
ELSE
	_buttonGroundLight.Reset();
END_IF
END_SET
END_PROPERTY

PROPERTY ButtonRecover : BOOL
GET
ButtonRecover := _buttonRecover._signal;
END_GET
SET
// Light up illumination of button
IF ButtonRecover THEN
	_buttonRecoverLight.Set();
ELSE
	_buttonRecoverLight.Reset();
END_IF
END_SET
END_PROPERTY

PROPERTY ButtonSuspend : BOOL
GET
ButtonSuspend := _buttonSuspend._signal;
END_GET
SET
// Light up illumination of button
IF ButtonSuspend THEN
	_buttonSuspendLight.Set();
ELSE
	_buttonSuspendLight.Reset();
END_IF
END_SET
END_PROPERTY

(*~
	<docu>
		<summary>
			Restores this instance to the Ready state. Can be called explicitly or from within one of the restore mechanisms.	
		</summary>			
	</docu>	
~*)
METHOD  Restore : ITcoRestorable
_buttonAutoLight.Reset();
_buttonGroundLight.Reset();
_buttonSuspendLight.Reset();
_buttonRecoverLight.Reset();
END_METHOD

(*~
	<docu>
		<summary>
		    Custom service (manual, maintenance) logic.
			This method must be implemented in derived class.
		</summary>			
	</docu>	
~*)
METHOD PROTECTED  ServiceMode
THIS^._buttonRecoverLight.Service();
THIS^._buttonSuspendLight.Service();
THIS^._buttonGroundLight.Service();
THIS^._buttonAutoLight.Service();
END_METHOD

END_FUNCTION_BLOCK

// ---- Abstractions/Safety/ControlledZone/TcoControlledZoneActionTask.TcPOU
FUNCTION_BLOCK PUBLIC  TcoControlledZoneActionTask EXTENDS TcoCore.TcoTask 
VAR_IN_OUT
	inoStatus:TcoControlledZone_Status;
END_VAR
VAR
    _progress : INT := 0;
    {attribute 'hide'} 
	_infoTimer :  TON;
    {attribute 'hide'} 
	_errorTimer :  TON;
    {attribute 'hide'} 
	_varInfo : __SYSTEM.VAR_INFO;
    {attribute 'hide'} 
	_sb : TcoCore.StringBuilder;

END_VAR

(*~
	<docu>
		<summary>
			Executes when task reaches the ```Done``` state .
		</summary>			
	</docu>	
~*)
METHOD PROTECTED OnDone
_progress := 0;
END_METHOD

PROPERTY PUBLIC Progress : REFERENCE TO INT
GET
Progress ref= _progress;
END_GET
END_PROPERTY

(*~
	<docu>
		<summary>
			Restores this instance to the Ready state. Can be called explicitly or from within one of the restore mechanisms.
			<para>
				See also <see cref="PlcDocu.TcoCore.TcoTask.AutoRestorable()"/>
			</para>
		</summary>			
	</docu>	
~*)
METHOD Restore : TcoCore.ITcoRestorable
SUPER^.Restore();
_progress := 0;
Messenger.UnPin();
END_METHOD

END_FUNCTION_BLOCK

// ---- Abstractions/Safety/ControlledZone/TcoControlledZone.TcPOU
FUNCTION_BLOCK TcoControlledZone EXTENDS TcoCore.TcoComponent
VAR_INPUT
	{attribute clr [RenderIgnore()]}
	inDoorCircuit        : ITcoDoorCircuit;
	
	{attribute clr [RenderIgnore()]}
	inAirPressureOK         : BOOL;
	
	{attribute clr [RenderIgnore()]}
	inEstopActive		      : BOOL;
	
END_VAR

VAR
	
	
	{attribute addProperty Name "<#Status#>"}
    {attribute clr [ReadOnly()]}
    _status : TcoControlledZone_Status;

	{attribute addProperty Name "<#Config#>"}
    _config : TcoControlledZone_Config;

	{attribute clr [RenderIgnore()]}
	_controlledUnits      : ARRAY [0..12] OF ICUBase;
				
	{attribute clr [RenderIgnore()]}
	_controlButtons       : ARRAY [0..4] OF ITcoControlButtons;
	
	{attribute clr [RenderIgnore()]}
	_controlKeyMode  : ARRAY [0..2] OF ITcoKeyMode;
	
	{attribute clr [RenderIgnore()]}
	_controlKeyNormalService      : ARRAY [0..2] OF ITcoKeyNormalSevice;
	
	// group states

	{attribute clr [RenderIgnore()]}
	_blinker              : TcoUtilities.TcoBlinker(THIS^);
	{attribute clr [RenderIgnore()]}
	_blinkerSlow              : TcoUtilities.TcoBlinker(THIS^);
	
	 {attribute addProperty Name "<#Ground task#>"}
	_groundTask           : TcoControlledZoneActionTask(THIS^);
	 {attribute addProperty Name "<#Automat task#>"}
	_autoTask           : TcoControlledZoneActionTask(THIS^);
	
	 {attribute addProperty Name "<#Recover task#>"}
	_recoverTask            : TcoControlledZoneActionTask(THIS^);
	
	 {attribute addProperty Name "<#Suspend task#>"}
	_suspendTask             : TcoControlledZoneActionTask(THIS^);
	
	 {attribute addProperty Name "<#Key Auto task#>"}
	_keyAutoTask          : TcoControlledZoneActionTask(THIS^);
	
	{attribute addProperty Name "<#Key Manual task#>"}
	_keyManualTask        : TcoControlledZoneActionTask(THIS^);
	
	{attribute addProperty Name "<#Key Step task#>"}
	_keyStepTask          : TcoControlledZoneActionTask(THIS^);
		
	 {attribute addProperty Name "<#Key service task#>"}
	_keyServiceTask             : TcoControlledZoneActionTask(THIS^);
	
	{attribute clr [RenderIgnore()]}
	_timerDoorsLocked       : TON;
	{attribute clr [RenderIgnore()]}
	_timerAirPressureMonitor       : TON;


	
	{attribute clr [RenderIgnore()]}
	_serviceKeyRising 	  : R_Trig;
	
	{attribute clr [RenderIgnore()]}
	_serviceKeyFalling 	  : F_Trig;
	
	
	{attribute clr [RenderIgnore()]}
	_recoverTaskInvokeFalling 	  : F_Trig;
	
	{attribute clr [RenderIgnore()]}
	_suspendTaskInvokeFalling 	  : F_Trig;
	
	{attribute clr [RenderIgnore()]}
	_recoverTaskInvokeRising 	  : R_Trig;
	
	{attribute clr [RenderIgnore()]}
	_suspendTaskInvokeRising 	  : R_Trig;
	
	{attribute clr [RenderIgnore()]}
	_groundTaskInvokeFalling 	  : F_Trig;

    {attribute clr [RenderIgnore()]}
	_autoTaskInvokeFalling 	  : F_Trig;
	
	{attribute clr [RenderIgnore()]}
	_groundTaskInvokeRising 	  : F_Trig;

    {attribute clr [RenderIgnore()]}
	_autoTaskInvokeRising 	  : F_Trig;
	
	{attribute clr [RenderIgnore()]}
	_keyAutoTaskInvokeFalling 	  : F_Trig;
	{attribute clr [RenderIgnore()]}
	_keyAutoTaskInvokeRising 	  : R_Trig;
	
	{attribute clr [RenderIgnore()]}
	_keyManualTaskInvokeFalling 	  : F_Trig;
	{attribute clr [RenderIgnore()]}
	_keyManualTaskInvokeRising 	  : R_Trig;
	
	{attribute clr [RenderIgnore()]}
	_keyStepTaskInvokeFalling 	  : F_Trig;
	{attribute clr [RenderIgnore()]}
	_keyStepTaskInvokeRising 	  : R_Trig;
	
	{attribute clr [RenderIgnore()]}
	_keyServiceTaskInvokeFalling 	  : F_Trig;
	{attribute clr [RenderIgnore()]}
	_keyServiceTaskInvokeRising 	  : R_Trig;

  
	_airPressureOk: BOOL;
	_conditionToRunAreSufficient: BOOL;
END_VAR

IF _controlledUnits[0] = 0 THEN
    THIS^.Messenger.Programming('<#Missing link to Controlled unit! No function is being executed!#>');
    RETURN;
END_IF

IF _controlButtons[0] = 0 
	OR _controlKeyMode[0] = 0 
	OR _controlKeyNormalService[0] = 0  THEN
    THIS^.Messenger.Programming('<#Missing link to control panel components (Buttons, Mode Keys, Normal/Service)! No function is being executed!#>');
    RETURN;
END_IF



_blinker(inOffTime := T#500MS, inOnTime := T#500MS);		//2 Hz
_blinkerSlow(inOffTime := T#1250MS, inOnTime := T#1250MS);	//0.8 Hz

THIS^.Initialize();

//presure monitoring
_airPressureOk:=TRUE;
_timerAirPressureMonitor(IN:=NOT inAirPressureOK,PT:=_config.AirPressureErrorTime);
IF _timerAirPressureMonitor.Q THEN
	_airPressureOk:=FALSE;
    THIS^.Messenger.Error('<#Air pressure is not sufficient!#>').Pin();
END_IF;

//Estop monitoring
IF THIS^.inEstopActive THEN
    inDoorCircuit.UnLock();
    THIS^.Messenger.Error('<#Emergency stop active: Unlocking doors!#>').Pin();
END_IF
// Global Voltage monitoring
IF NOT inDoorCircuit.IsGlobalVoltageOk THEN
    inDoorCircuit.UnLock();
    THIS^.Messenger.Error('<#Global control voltage interrupted: Unlocking doors!#>').Pin();
END_IF

//Voltage monitoring todo
_timerDoorsLocked(IN := inDoorCircuit.IsClosed AND inDoorCircuit.IsLocked AND  inDoorCircuit.IsLocalDoorsVoltageOk, PT := _config.DoorsLocked);

IF _timerDoorsLocked.Q THEN
    IF NOT inDoorCircuit.IsLocalVoltageOk THEN
        // unlock doors in case that control voltage goes down and it shouldn't
        inDoorCircuit.UnLock();
        THIS^.Messenger.Error('<#Local voltage interrupted: Unlocking doors!#>');
    END_IF
END_IF


_conditionToRunAreSufficient:=(inAirPressureOK OR _timerAirPressureMonitor.ET<_timerAirPressureMonitor.PT) AND NOT inEstopActive  AND inDoorCircuit.IsGlobalVoltageOk AND inDoorCircuit.IsLocalVoltageOk;
 


_recoverTaskInvokeRising(CLK:=_status.State.AnyButtonRecover);
_recoverTaskInvokeFalling(CLK:=_status.State.AnyButtonRecover);
IF _recoverTaskInvokeRising.Q THEN
	_recoverTask.Restore();
END_IF
IF _recoverTaskInvokeFalling.Q THEN
	_recoverTask.Invoke();
	_suspendTask.Restore();
END_IF



_suspendTaskInvokeRising(CLK:=_status.State.AnyButtonSuspend);
_suspendTaskInvokeFalling(CLK:=_status.State.AnyButtonSuspend);
IF _suspendTaskInvokeRising.Q THEN
	_suspendTask.Restore();
END_IF
IF _suspendTaskInvokeFalling.Q THEN
	_suspendTask.Invoke();
	_recoverTask.Restore();
END_IF





_groundTaskInvokeRising(CLK:=_status.State.AnyButtonGround);
IF _groundTaskInvokeRising.Q THEN
	_groundTask.Restore();
END_IF
_groundTaskInvokeFalling(CLK:=_status.State.AnyButtonGround);
IF _groundTaskInvokeFalling.Q THEN
	_groundTask.Invoke();
END_IF
_groundTask.Enabled:= (_conditionToRunAreSufficient
						AND inDoorCircuit.IsLocalDoorsVoltageOk 
						AND _status.State.AllKeysAuto 
						AND _status.State.AllKeysNormal) ;

IF _groundTask.Busy THEN
	_autoTask.Restore();
END_IF						
						
_autoTaskInvokeRising(CLK:=_status.State.AnyButtonAuto);
IF _autoTaskInvokeRising.Q THEN
	_autoTask.Restore();
END_IF

_autoTaskInvokeFalling(CLK:=_status.State.AnyButtonAuto);
IF _autoTaskInvokeFalling.Q THEN
	_autoTask.Invoke();
END_IF

_autoTask.Enabled:= (_conditionToRunAreSufficient 
					AND inDoorCircuit.IsLocalDoorsVoltageOk 
					AND _status.State.AllKeysAuto 
					AND _status.State.AllKeysNormal) ;





//----------keys -----------

// key auto
_keyAutoTaskInvokeFalling(CLK:= _status.State.AllKeysAuto);
_keyAutoTaskInvokeRising(CLK:=_status.State.AllKeysAuto);

IF _keyAutoTaskInvokeRising.Q THEN
	_keyAutoTask.Invoke();
END_IF
IF _keyAutoTaskInvokeFalling.Q THEN
	_keyAutoTask.Restore();
END_IF


// key manual
_keyManualTaskInvokeRising(CLK:= _status.State.AnyKeyManual);
_keyManualTaskInvokeFalling(CLK:=_status.State.AnyKeyManual);

IF _keyManualTaskInvokeRising.Q THEN
	_keyManualTask.Invoke();
END_IF
IF _keyManualTaskInvokeFalling.Q THEN
	_keyManualTask.Restore();
END_IF


IF _status.State.AnyKeyStep AND _keyStepTask.Ready THEN
	_keyStepTask.Invoke();
END_IF
IF _status.State.AnyKeyStep AND _keyStepTask.Done THEN
	_keyStepTask.Restore();
END_IF

_keyStepTaskInvokeFalling(CLK:=_status.State.AnyKeyStep);

IF _keyStepTaskInvokeFalling.Q THEN
	_keyStepTask.Restore();
END_IF


// key service
_keyServiceTaskInvokeRising(CLK:= _status.State.AnyKeyService);
_keyServiceTaskInvokeFalling(CLK:=_status.State.AnyKeyService);

IF _keyServiceTaskInvokeRising.Q THEN
	_keyServiceTask.Invoke();
END_IF
IF _keyServiceTaskInvokeFalling.Q THEN
	_keyServiceTask.Restore();
END_IF






// Handling of buttons
THIS^.ButtonRecover();
THIS^.ButtonSuspend();
THIS^.ButtonGround();
THIS^.ButtonAuto();


// Handling of key 1
THIS^.KeyAuto();
THIS^.KeyManual();
THIS^.KeyStep();

// Handling of Key Normal/Service
THIS^.KeyService();

METHOD AddControlButtons : BOOL
VAR_INPUT
 	inControlButtons : ITcoControlButtons;
END_VAR
VAR
	i : UINT;
END_VAR
AddControlButtons := FALSE;

IF inControlButtons = 0 THEN
	RETURN;
END_IF

FOR i := 0 TO _config.MaxControlButtons DO
	IF _controlButtons[i] = inControlButtons THEN
		AddControlButtons := TRUE;
		RETURN;
	END_IF
	
	IF 	_controlButtons[i] = 0 THEN
		_controlButtons[i] := inControlButtons;
		AddControlButtons  := TRUE;
		RETURN;
	END_IF
END_FOR
END_METHOD

METHOD AddControlledUnit : BOOL
VAR_INPUT
 	inControlledUnit : ICUBase;
END_VAR
VAR
	i : UINT;
END_VAR
AddControlledUnit := FALSE;

IF inControlledUnit = 0 THEN
	RETURN;
END_IF

FOR i := 0 TO _config.MaxControledUnits DO
	IF _controlledUnits[i] = inControlledUnit THEN
		AddControlledUnit := TRUE;
		RETURN;
	END_IF
	
	IF 	_controlledUnits[i] = 0 THEN
		_controlledUnits[i] := inControlledUnit;
		AddControlledUnit    := TRUE;
		RETURN;
	END_IF
END_FOR
END_METHOD

METHOD AddKeyMode : BOOL
VAR_INPUT
 	inKeyMode : ITcoKeyMode;
END_VAR
VAR
	i : UINT;
END_VAR
AddKeyMode := FALSE;

IF inKeyMode = 0 THEN
	RETURN;
END_IF

FOR i := 0 TO  _config.MaxKeyMode DO
	IF _controlKeyMode[i] = inKeyMode THEN
		AddKeyMode := TRUE;
		RETURN;
	END_IF
	
	IF 	_controlKeyMode[i] = 0 THEN
		_controlKeyMode[i] := inKeyMode;
		AddKeyMode    := TRUE;
		RETURN;
	END_IF
END_FOR
END_METHOD

METHOD AddKeyNormalService : BOOL
VAR_INPUT
 	inKeyNormalService : ITcoKeyNormalSevice;
END_VAR
VAR
	i : UINT;
END_VAR
AddKeyNormalService := FALSE;

IF inKeyNormalService = 0 THEN
	RETURN;
END_IF

FOR i := 0 TO _config.MaxKeyNormalService DO
	IF _controlKeyNormalService[i] = inKeyNormalService THEN
		AddKeyNormalService := TRUE;
		RETURN;
	END_IF
	
	IF 	_controlKeyNormalService[i] = 0 THEN
		_controlKeyNormalService[i] := inKeyNormalService;
		AddKeyNormalService    := TRUE;
		RETURN;
	END_IF
END_FOR
END_METHOD

PROPERTY PUBLIC AirPressureOk : bool
GET
AirPressureOk:=_airPressureOk;
END_GET
END_PROPERTY

{attribute 'monitoring' := 'variable'}
PROPERTY AnyButtonAuto : BOOL
GET
AnyButtonAuto := _status.State.AnyButtonAuto;
END_GET
SET
VAR
	button : UINT;
END_VAR
FOR button := 0 TO _config.MaxControlButtons DO
	IF _controlButtons[button] <> 0 THEN
		_controlButtons[button].ButtonAuto := AnyButtonAuto;
	ELSE
		EXIT;
	END_IF
END_FOR
END_SET
END_PROPERTY

{attribute 'monitoring' := 'variable'}
PROPERTY AnyButtonGround : BOOL
GET
AnyButtonGround := _Status.State.AnyButtonGround;
END_GET
SET
VAR
	button : UINT;
END_VAR
FOR button := 0 TO _config.MaxControlButtons DO
	IF _controlButtons[button] <> 0 THEN
		_controlButtons[button].ButtonGround := AnyButtonGround;
	ELSE
		EXIT;
	END_IF
END_FOR
END_SET
END_PROPERTY

{attribute 'monitoring' := 'variable'}
PROPERTY AnyButtonRecover : BOOL
GET
AnyButtonRecover := _status.State.AnyButtonRecover;
END_GET
SET
VAR
	button : UINT;
END_VAR
FOR button := 0 TO _config.MaxControlButtons DO
	IF _controlButtons[button] <> 0 THEN
		_controlButtons[button].ButtonRecover := AnyButtonRecover;
	ELSE
		EXIT;
	END_IF
END_FOR
END_SET
END_PROPERTY

{attribute 'monitoring' := 'variable'}
PROPERTY AnyButtonSuspend : BOOL
GET
AnyButtonSuspend := _status.State.AnyButtonSuspend;
END_GET
SET
VAR
	button : UINT;
END_VAR
FOR button := 0 TO _config.MaxControlButtons DO
	IF _controlButtons[button] <> 0 THEN
		_controlButtons[button].ButtonSuspend := AnyButtonSuspend;
	ELSE
		EXIT;
	END_IF
END_FOR
END_SET
END_PROPERTY

METHOD ButtonAuto : BOOL
VAR
	cu : UINT;
END_VAR


IF _autoTask.Execute() THEN
	AnyButtonGround:=FALSE;
	AnyButtonAuto:=_blinkerSlow.IsOn ;		

	IF _autoTask.Progress =0 THEN
	
		IF 	_status.State.AllKeysAuto AND _status.State.AllKeysNormal  THEN
	
			_status.ActionDescription:= '<#Automat mode has been invoked.#>';
			FOR cu := 0 TO _config.MaxControledUnits DO
				IF _controlledUnits[cu] <> 0 THEN
					IF   _controlledUnits[cu].StatusInfo.Mode = eCUMode.GroundModeDone    THEN
						_controlledUnits[cu].AutomatTask.Task.Invoke();
					END_IF	
	
					IF _controlledUnits[cu].StatusInfo.Mode=eCUMode.AutomatMode THEN
							_controlledUnits[cu].AutomatTask.ModeController.Mode:=eSequencerMode.CyclicMode;	
					End_if;	
				ELSE
					EXIT;
				END_IF
			END_FOR
			_autoTask.Progress := _autoTask.Progress + 1;	
			RETURN;
		ELSE
			_status.ActionDescription:= '<#Mode keys are not in correct position.#>';
		END_IF;
			
	ELSE
		
		_autoTask.DoneWhen(_status.State.AllInAuto AND NOT _status.State.AnyButtonAuto);	
		 IF _autoTask.Done THEN
			 
		 	_status.ActionDescription:= '<#Automat mode has been done.#>';
			AnyButtonAuto:=TRUE;
		END_IF;	
	END_IF;
	
	IF _status.ActionDescription<>'' THEN
		THIS^._autoTask.Messenger.Notify(_status.ActionDescription);
	END_IF;
END_IF;
END_METHOD

METHOD ButtonGround : BOOL
VAR
	cu : UINT;
END_VAR

IF _groundTask.Execute() THEN
	// led signalisation
	AnyButtonAuto:=FALSE;
	AnyButtonGround:=_blinkerSlow.IsOn ;	

	IF _groundTask.Progress =0 THEN
		IF 	_status.State.AllKeysAuto AND _status.State.AllKeysNormal  THEN
	
			_status.ActionDescription:= '<#Grounding mode has been invoked.#>';
			FOR cu := 0 TO _config.MaxControledUnits DO
				IF _controlledUnits[cu] <> 0 THEN
					IF  _controlledUnits[cu].StatusInfo.Mode<> eCUMode.GroundMode OR _controlledUnits[cu].StatusInfo.Mode<> eCUMode.GroundModeDone THEN
						_controlledUnits[cu].GroundTask.Task.Invoke();
					END_IF	
					IF _controlledUnits[cu].StatusInfo.Mode=eCUMode.GroundMode THEN
							_controlledUnits[cu].GroundTask.ModeController.Mode:=eSequencerMode.CyclicMode;	
					End_if;			
				ELSE
					EXIT;
				END_IF
			END_FOR
			
			_groundTask.Progress := _groundTask.Progress + 1;	
			RETURN;
		ELSE
			_status.ActionDescription:= '<#Mode keys are not in correct position.#>';
		END_IF;
		
	ELSE
		
		_groundTask.DoneWhen(_status.State.AllGrounded AND NOT _status.State.AnyButtonGround );	
		 IF _groundTask.Done THEN
			 _status.ActionDescription:= '<#Grounding mode has been done.#>';
			AnyButtonGround:=TRUE;
		END_IF;	
	END_IF	
	IF _status.ActionDescription<>'' THEN
		THIS^._groundTask.Messenger.Notify(_status.ActionDescription);
	END_IF;
	

END_IF;
END_METHOD

METHOD ButtonRecover : BOOL
VAR
	cu : UINT;
END_VAR

IF _recoverTask.Execute() THEN
	AnyButtonSuspend:=FALSE;

	IF _recoverTask.Progress = 2 THEN
		AnyButtonRecover:=_blinker.IsOn ;
	ELSE
		AnyButtonRecover:=_blinkerSlow.IsOn ;	
	END_IF;
	IF _recoverTask.Progress =0 THEN
		FOR cu := 0 TO _config.MaxControledUnits DO
			IF _controlledUnits[cu] <> 0 THEN
				_controlledUnits[cu].RecoverTask.Restore();
			ELSE
				EXIT;
			END_IF
		END_FOR

		_status.ActionDescription:='<#Waiting to release recover button#>';
		IF NOT _status.State.AnyButtonRecover THEN
				_recoverTask.Progress := _recoverTask.Progress + 1;	
				RETURN;
		END_IF;
	
	END_IF
	
	IF _recoverTask.Progress =1 THEN
		_status.ActionDescription:='<#Check general condition to recover zone (ControlVoltage, EStops, Presure...)!#>';
				
		IF inDoorCircuit.IsGlobalVoltageOk
			AND inDoorCircuit.IsLocalVoltageOk
			AND inAirPressureOK
			AND NOT inEstopActive THEN
			_recoverTask.Progress := _recoverTask.Progress + 1;
	
		END_IF;
	
	END_IF
	
	IF _recoverTask.Progress =2 THEN
		_status.ActionDescription:='<#Waiting to close and lock  all doors!#>';
		
		THIS^.inDoorCircuit.Lock();
		
			
		IF inDoorCircuit.IsLocked
			AND inDoorCircuit.IsLocked
			AND inDoorCircuit.IsLocalDoorsVoltageOk THEN
			_recoverTask.Progress := _recoverTask.Progress + 1;
	
		END_IF;
	
	END_IF


	
	
	IF _recoverTask.Progress =3 THEN
		
		_status.ActionDescription:='<#Invoke restore sequences on each stations.#>';
		IF _status.State.AllInManual OR _status.State.AllInactiveOrManualOrGrounded THEN
			_recoverTask.Progress := 100;
			RETURN;
		END_IF
		
		FOR cu := 0 TO _config.MaxControledUnits DO
			IF _controlledUnits[cu] <> 0 THEN
				_controlledUnits[cu].RecoverTask.ModeController.Mode := eSequencerMode.CyclicMode;
				_controlledUnits[cu].RecoverTask.Task.Invoke();

			ELSE
				EXIT;
			END_IF
		END_FOR

		IF _status.State.AllRecovered THEN
			_recoverTask.Progress :=_recoverTask.Progress+1 ;
		END_IF
		
	END_IF
	
	IF _recoverTask.Progress =4 THEN
		
		_status.ActionDescription:= '<#Setup Cyclic or Step mode. It depends on key position#>';
		FOR cu := 0 TO _config.MaxControledUnits DO
			IF _controlledUnits[cu] <> 0 THEN
				IF _status.State.AllKeysAuto THEN	
					IF _controlledUnits[cu].StatusInfo.Mode=eCUMode.AutomatMode THEN
						_controlledUnits[cu].AutomatTask.ModeController.Mode:=eSequencerMode.CyclicMode;
					ELSIF _controlledUnits[cu].StatusInfo.Mode=eCUMode.GroundMode THEN
						_controlledUnits[cu].GroundTask.ModeController.Mode:=eSequencerMode.CyclicMode;
					END_IF
				ELSE
					IF _controlledUnits[cu].StatusInfo.Mode=eCUMode.AutomatMode THEN
						_controlledUnits[cu].AutomatTask.ModeController.Mode:=eSequencerMode.StepMode;
					ELSIF _controlledUnits[cu].StatusInfo.Mode=eCUMode.GroundMode THEN
						_controlledUnits[cu].GroundTask.ModeController.Mode:=eSequencerMode.StepMode;
					END_IF
				END_IF
	
			ELSE
				EXIT;
			END_IF
		END_FOR


		
		
		_recoverTask.Progress := 100;
		
	END_IF

	IF _recoverTask.Progress = 100 THEN
		
		_status.ActionDescription:= '<#Recover task has been done.#>';
		_recoverTask.DoneWhen(TRUE);
		AnyButtonRecover:=TRUE;

	END_IF;	


	IF _status.ActionDescription<>'' THEN
		THIS^._recoverTask.Messenger.Notify(_status.ActionDescription);
	END_IF;
	
END_IF;
END_METHOD

METHOD ButtonSuspend : BOOL
VAR
	cu : UINT;
END_VAR
IF _suspendTask.Execute() THEN
	AnyButtonRecover:=FALSE;
	AnyButtonSuspend:=_blinkerSlow.IsOn ;	
	IF _suspendTask.Progress =0 THEN
		FOR cu := 0 TO _config.MaxControledUnits DO
			IF _controlledUnits[cu] <> 0 THEN
				_controlledUnits[cu].SuspendTask.Restore();

			ELSE
				EXIT;
			END_IF
		END_FOR
		_status.ActionDescription:='<#Waiting to release suspend button#>';
		IF NOT _status.State.AnyButtonSuspend THEN
				_suspendTask.Progress := _suspendTask.Progress + 1;	
				RETURN;

		END_IF;
	
	END_IF
	
	IF _suspendTask.Progress =1 THEN
		_status.ActionDescription:='<#Check general condition to suspned zone (ControlVoltage,EStops,Presure...)!#>';
		
		IF NOT inDoorCircuit.IsGlobalVoltageOk
			OR NOT inDoorCircuit.IsLocalVoltageOk
			OR NOT inAirPressureOK
			OR inEstopActive THEN
			_suspendTask.Progress := 100;
			
			THIS^.inDoorCircuit.Unlock();
		ELSE
			_suspendTask.Progress := _suspendTask.Progress + 1;	
		END_IF;
	
	END_IF
	
	IF _suspendTask.Progress =2 THEN
		
		_status.ActionDescription:= '<#Force step mode.#>';
		
		IF _status.State.AllInManual OR _status.State.AllInactiveOrManualOrGrounded THEN
			_suspendTask.Progress := 100;
			RETURN;
		END_IF
		FOR cu := 0 TO _config.MaxControledUnits DO
			IF _controlledUnits[cu] <> 0 THEN
			

				IF _controlledUnits[cu].StatusInfo.Mode=eCUMode.AutomatMode THEN
					_controlledUnits[cu].AutomatTask.ModeController.Mode:=eSequencerMode.StepMode;
				ELSIF _controlledUnits[cu].StatusInfo.Mode=eCUMode.GroundMode THEN
					_controlledUnits[cu].GroundTask.ModeController.Mode:=eSequencerMode.StepMode;
				END_IF
		
	
			ELSE
				EXIT;
			END_IF
		END_FOR


		
		IF _status.State.AllInStepMode THEN
			_suspendTask.Progress := _suspendTask.Progress + 1;
		END_IF;
			
	END_IF
	
	IF _suspendTask.Progress =3 THEN
		
		_status.ActionDescription:='<#Invoke suspend sequences on each stations.#>';
		
		
		FOR cu := 0 TO _config.MaxControledUnits DO
			IF _controlledUnits[cu] <> 0 THEN
				_controlledUnits[cu].SuspendTask.ModeController.Mode := eSequencerMode.CyclicMode;
				_controlledUnits[cu].SuspendTask.Task.Invoke();

			ELSE
				EXIT;
			END_IF
		END_FOR

		IF _status.State.AllSuspended THEN
			_suspendTask.Progress := _suspendTask.Progress+1;
		END_IF
		
	END_IF
	
	
	
	IF _suspendTask.Progress =4 THEN
		_status.ActionDescription:='<#Waiting to unlock  all doors!#>';
		
		THIS^.inDoorCircuit.UnLock();
		
		IF inDoorCircuit.IsUnLocked THEN
			_suspendTask.Progress := 100;
	
		END_IF;
	
	END_IF


	IF _suspendTask.Progress = 100 THEN
		_status.ActionDescription:= '<#Suspend task has been done.#>';
		_suspendTask.DoneWhen(TRUE);
		AnyButtonSuspend:=TRUE;
	END_IF;	


	IF _status.ActionDescription<>'' THEN
		THIS^._suspendTask.Messenger.Notify(_status.ActionDescription);
	END_IF;
	
END_IF;
END_METHOD

PROPERTY Config :REFERENCE TO TcoControlledZone_Config
GET
Config ref=_config;
END_GET
END_PROPERTY

METHOD Initialize : BOOL
VAR
	i : UINT;

END_VAR
_status.State.AllInAuto := TRUE;
_status.State.AllInGrounding := TRUE;
_status.State.AllInManual := TRUE;
_status.State.AllIdle := TRUE;
_status.State.AllGrounded := TRUE;
_status.State.AllInStepMode := TRUE;
_status.State.AllSuspended := TRUE;
_status.State.AllRecovered := TRUE;
_status.State.AllInactiveOrManualOrGrounded :=true;
_status.State.AnyInAuto := FALSE;
_status.State.AnyInManual := FALSE;
_status.State.AnyGrounding := FALSE;
_status.State.AnyInStepMode := FALSE;

i := 0;

